	// Hier zum BMK noch die Ist-Position hinzufügen. Die Ist-Position wünschte sich nobilia. Das BMK bietet sich dafür an. Weitere Variablen in die Meldestruktur ist nicht möglich.
	IF IQ_stAchse.stMeldg.bEndlPosAngf
		OR bTestMeldAchs
	THEN
		IQ_stUniAnstgHMI.stAchsMeldHMI.sBMK :=
			CONCAT(I_sAktorBMK,
			CONCAT(' Istposition: ',TO_STRING(IQ_stAchse.fPosIstwert)));
	END_IF

	IQ_stUniAnstgHMI.stAchsMeldHMI.bMeldEndlPos				:= IQ_stAchse.stMeldg.bEndlPosAngf
																				OR bTestMeldAchs;			

	(**************************************************)
END_ACTION

END_FUNCTION_BLOCK

// POUs/UniBausteine/FB_UniAktrAnstg
(*
Beschreibung :	UniFB zur Hardwaresteuerung, Anzeige und Fehlermeldung in der Avalon HMI eines allgemeinen Aktors
					mit einem Überwachungseingang/Rückmeldung, ob auch eingeschaltet wurde.
					inkl. Handling - Handfunktinen
										- Meldefunktionen
										- Betriebsarten
										- Schutzbereiche
					Datentypen: ST_UniBaustein
									ST_UniAktrAnstg
					Ressourcen: GlobalVar_Allgemein
									GlobalVar_Farben
									AllgemeineParameter
TwinCat Vers.:	3.1.4024.25							
Erstellt		 :	Anlagentechnik Grp.11 (BECKHOFF AUTOMATION)
*)
FUNCTION_BLOCK FB_UniAktrAnstg
VAR_INPUT

	I_sStatName			:Tc2_System.T_MaxString;	// Aktueller Stationsname
	I_sAktorName		:Tc2_System.T_MaxString;	// Aktueller Aktorname von der Funktion des Aktors
	I_sAktorBMK1		:Tc2_System.T_MaxString;	// BMK - Rückmeldung

	I_bResHandFkt		:BOOL;	// Funktion-Reset für Grundstellungsablauf
	I_bZuwGrdstFkt		:BOOL;	// Funktion-Zuweisung Grundstellungsablauf
	I_bZuwAutomFkt		:BOOL;	// Funktion-Zuweisung Automatikablauf

	I_bAktrAbfrg		:BOOL;	// Abfrage z.B. Vakuum aufgebaut

	I_nSchutzBer		:INT;		// Schutzbereich => Betriebsart

	(*Optionale Funktionen*)													
	I_bResHdBetr		:BOOL;	// Ausschalten des Aktors beim Wechsel auf Handbetrieb
																						
	I_tLaufzVorg		:TIME:= T#5S;	(*Angepasste Meldelaufzeit*)	
	I_bVerrMeldg		:BOOL;	(*Meldungsausgabe Unterdrücken*)
																						
	I_bAnstgUng			:BOOL;	(*Ansteuerung Ungeschaltet*)	
	I_bAnstgInvt		:BOOL;	(*Ansteuerung Invertieren*)
	I_eAnstgDef			:E_AnstgArtUniAktr := eAktrAusEinschalt;	// Definition der Meldetexte und Anzeigetexte.
	
	I_sZuDef0			:Tc2_System.T_MaxString;	// eigene Definition für die linke Tasterbeschriftung
	I_sInDef0			:Tc2_System.T_MaxString;	// eigene Definition für die linke Tasterbeschriftung
	I_sZuDef1			:Tc2_System.T_MaxString;	// eigene Definition für die rechte Tasterbeschriftung
	I_sInDef1			:Tc2_System.T_MaxString;	// eigene Definition für die rechte Tasterbeschriftung

	I_stVarInfoBMK		:__SYSTEM.VAR_INFO;	// Optional: __VARINFO von einem Hardwareeingang. Kann I_sAktorBMK1 ersetzen. I_sAktorBMK1 ist aber dominant. Nicht im Aufruf verwenden => separate Zuweisung
END_VAR
VAR_IN_OUT

	IQ_stUniAnstgHMI	:ST_UniAktrAnstg;	// HMI-Strukturen

END_VAR
VAR_OUTPUT

	Q_bAktrAnstg		:BOOL;	// Ansteuerung z.B. Sauger Ein

END_VAR
VAR

	sTextHandFkt1		:ARRAY[0..1] OF STRING(20);				
	sTextHandFkt2		:ARRAY[0..1] OF STRING(20);					
	sTextHandFktX		:ARRAY[0..1] OF STRING(20);	// Zum Zwischenspeichern

	fbLfzMeldAusg		:FB_LaufzMeldgAktr;

	//Relevante Variablen zur Diagnose
	stUniAnstgFkt		:ST_UniBaustein;
END_VAR

	(*Uni.- Aktorenansteuerung*)
	
	(**************************************************)	
	(*Aufruf-Bereichskontrolle*)

	IF I_nSchutzBer <= 0 OR I_nSchutzBer > cAnzSchutzBer
		THEN
			IQ_stUniAnstgHMI.stMeldAusgHMI.sMeldText		:= 'I_nSchutzBer = 0 oder zu gross.';
			IQ_stUniAnstgHMI.stMeldAusgHMI.SourceName		:= I_sStatName;
			IQ_stUniAnstgHMI.stMeldAusgHMI.sAktorName		:= I_sAktorName;

			IF I_sAktorBMK1 <> ''
			THEN	// I_sAktorBMK1 ist beschrieben. Damit wird der String als BMK genommen
				IQ_stUniAnstgHMI.stMeldAusgHMI.sBMK	:= I_sAktorBMK1;
			ELSE	// Der Kommentar von VARINFO wird als BMK genommen
				IQ_stUniAnstgHMI.stMeldAusgHMI.sBMK	:= I_stVarInfoBMK.Comment;
			END_IF
			
			IQ_stUniAnstgHMI.stMeldAusgHMI.bMeldHinweis	:= TRUE;
			stUniAnstgFkt.nHandStat:= 256;	// Funktion sperren
			y_ZustAnzg();
			RETURN;
		ELSE
			IQ_stUniAnstgHMI.stMeldAusgHMI.bMeldHinweis	:= FALSE;
			IQ_stUniAnstgHMI.stMeldAusgHMI.sMeldText		:= '';
	END_IF

	(**************************************************)	
	(*Haendling Uni-Struktur*)

	a_Standard();

	(**************************************************)	
	(*Ausgänge zuweisen*)

	x_AusgZuw();
	
	(**************************************************)	
	(*Zustände anzeigen*)

	y_ZustAnzg();

	(**************************************************)	
	(*Meldungen ausgeben*)

	z_FehlMeld();
	
	(**************************************************)

ACTION a_Standard:
	(*Ansteuerungstyp "Standard" /z.B. Vakuumsauger...*)

	(*Verwendete Softkeytasten = 2 (s.Beispiel)*)

   (*       "Handfunktion"       /   "Softkeytaste 1"   /   "Softkeytaste 2"   *)
	(*                                                                          *) 
   (*------- Vakuumeinheit ------/_____ausschalten______/_____einschalten______*)
	
	(*Softkeyleiste.1		:Funktion ausschalten*)
	(*Softkeyleiste.2		:Funktion einschalten*)

	(*Hinweis:
	- Funktion wird durch "ResHdBetr" bei Betriebsartenwechsel zurückgenommen
	
	- Mit "LaufzVorg" kann die Meldelaufzeit angepasst werden (Default: 5sek)
	- Mit "VerrMeldg" wird die Meldeausgabe unterdrückt (eventl. Ablaufbedingt)
	
	- Bei "AnstgUng" bleiben die F-Ausgänge auch bei geöffn. Schutzbereich aktiv  
	- Bei "AnstgInvt" wird die Logik der Funktions-Ausgänge invertiert  
	*)

	(**************************************************)	

	stUniAnstgFkt.bHandAnw0:= IQ_stUniAnstgHMI.stHandFktHMI[1].bySwitch > 0;
	stUniAnstgFkt.bHandAnw1:= IQ_stUniAnstgHMI.stHandFktHMI[2].bySwitch > 0;
	
	IF arrBetrartAutomAktiv[I_nSchutzBer]
		OR I_bResHandFkt
		THEN
			stUniAnstgFkt.arrHandFkt[1]:= FALSE;
		ELSE
			IF arrBetrartAutomSpeichn[I_nSchutzBer]
				THEN
					IF NOT I_bResHdBetr THEN
						stUniAnstgFkt.arrHandFkt[1]:= stUniAnstgFkt.arrFktAusfg[1];
					END_IF
				ELSE
					IF NOT arrGrdstlgBetrAktiv[I_nSchutzBer]
						AND arrBetrartHandAktiv[I_nSchutzBer]
						THEN
							 IF stUniAnstgFkt.bHandAnw1 THEN
								 stUniAnstgFkt.arrHandFkt[1]:= TRUE;
							 END_IF
							 IF stUniAnstgFkt.bHandAnw0 THEN
								 stUniAnstgFkt.arrHandFkt[1]:= FALSE;
							 END_IF
					END_IF
			END_IF
	END_IF

	IF arrBetrartHandAktiv[I_nSchutzBer]
		THEN
			IF stUniAnstgFkt.arrHandFkt[1]
				THEN
					stUniAnstgFkt.nHandStat:= 2;	(*Handfunktion.2 aktiv*)
				ELSE
					stUniAnstgFkt.nHandStat:= 1;	(*Handfunktion.1 aktiv*)
			END_IF
		ELSE
			stUniAnstgFkt.nHandStat:= 256;		(*Funktion gesperrt*)
	END_IF

	(**************************************************)	

	IF arrBetrartHandAktiv[I_nSchutzBer]
		THEN
			stUniAnstgFkt.arrGrdstFkt[1]:= I_bZuwGrdstFkt;
		ELSE
			stUniAnstgFkt.arrGrdstFkt[1]:= FALSE;
   END_IF
	IF arrBetrartAutomAktiv[I_nSchutzBer] OR TRUE //ToDo
		THEN
			stUniAnstgFkt.arrAutomFkt[1]:= I_bZuwAutomFkt;
		ELSE
			stUniAnstgFkt.arrAutomFkt[1]:= FALSE;
   END_IF

	(**************************************************)	

	stUniAnstgFkt.arrFktAusfg[1]:= stUniAnstgFkt.arrGrdstFkt[1]
										  	 OR stUniAnstgFkt.arrHandFkt[1]
										    OR stUniAnstgFkt.arrAutomFkt[1];

	(**************************************************)
END_ACTION

ACTION x_AusgZuw:

	(**************************************************)	
	(*Ausgänge zuweisen*)

	Q_bAktrAnstg:= stUniAnstgFkt.arrFktAusfg[1]
					 	AND (arrAusgGruppeFrg[I_nSchutzBer]
				    	OR I_bAnstgUng)
					 	AND bVersEingAusgAnlagOk;

	(**************************************************)	
	(*Ausgänge invertieren*)

	IF I_bAnstgInvt THEN
		Q_bAktrAnstg:= NOT Q_bAktrAnstg;
	END_IF

	(**************************************************)
END_ACTION

ACTION y_ZustAnzg:
	
	(**************************************************)	
	(*Zustände anzeigen*)
	CASE I_eAnstgDef OF
eAktrDef0Def1,
eAktrDef1Def0:
						sTextHandFkt1[0]:= I_sZuDef0;
						sTextHandFkt1[1]:= I_sInDef0;
						sTextHandFkt2[0]:= I_sZuDef1;
						sTextHandFkt2[1]:= I_sInDef1;
	
eAktrAusEinschalt,
eAktrEinAusschalt:
						sTextHandFkt1[0]:= 'einschalten';
						sTextHandFkt1[1]:= 'eingeschaltet';
						sTextHandFkt2[0]:= 'ausschalten';
						sTextHandFkt2[1]:= 'ausgeschaltet';
eAktrAusEinfahr,
eAktrEinAusfahr:
						sTextHandFkt1[0]:= 'einfahren';
						sTextHandFkt1[1]:= 'eingefahren';
						sTextHandFkt2[0]:= 'ausfahren';
						sTextHandFkt2[1]:= 'ausgefahren';
eAktrHebenSenken,
eAktrSenkenHeben:
						sTextHandFkt1[0]:= 'senken';
						sTextHandFkt1[1]:= 'abgesenkt';
						sTextHandFkt2[0]:= 'heben';
						sTextHandFkt2[1]:= 'angehoben';
	END_CASE
	
	IF I_eAnstgDef >= 20 //Zuweisungen tauschen 
		THEN
			sTextHandFktX:= sTextHandFkt1; 
			sTextHandFkt1:= sTextHandFkt2;
			sTextHandFkt2:= sTextHandFktX;
	END_IF
	
	IF stUniAnstgFkt.nHandStat = 1	(*Handfunktion.1 aktiv*)
		THEN
			IQ_stUniAnstgHMI.stHandFktHMI[1].sColour:= cGruenAsString;
			IQ_stUniAnstgHMI.stHandFktHMI[1].sText:= sTextHandFkt1[1];
		ELSE
			IQ_stUniAnstgHMI.stHandFktHMI[1].sColour:= cDefaultAsString;
			IQ_stUniAnstgHMI.stHandFktHMI[1].sText:= sTextHandFkt1[0];
   END_IF
	IF stUniAnstgFkt.nHandStat = 2	(*Handfunktion.2 aktiv*)
		THEN		 
			IQ_stUniAnstgHMI.stHandFktHMI[2].sColour:= cGruenAsString;
			IQ_stUniAnstgHMI.stHandFktHMI[2].sText:= sTextHandFkt2[1];
		ELSE
			IQ_stUniAnstgHMI.stHandFktHMI[2].sColour:= cDefaultAsString;
			IQ_stUniAnstgHMI.stHandFktHMI[2].sText:= sTextHandFkt2[0];
   END_IF
	IF stUniAnstgFkt.nHandStat = 256	(*Funktion gesperrt*)
		THEN
			IQ_stUniAnstgHMI.stHandFktHMI[1].byStatus:=
			IQ_stUniAnstgHMI.stHandFktHMI[2].byStatus:= 1;
			IQ_stUniAnstgHMI.stHandFktHMI[1].sText:= sTextHandFkt1[0];
			IQ_stUniAnstgHMI.stHandFktHMI[2].sText:= sTextHandFkt2[0];
		ELSE
			IQ_stUniAnstgHMI.stHandFktHMI[1].byStatus:=
			IQ_stUniAnstgHMI.stHandFktHMI[2].byStatus:= 0;
   END_IF

	(**************************************************)
END_ACTION

ACTION z_FehlMeld:

	(**************************************************)	
	(*Meldungen ausgeben*)

	fbLfzMeldAusg.I_bLaufzAnstg1:=	(Q_bAktrAnstg
													AND NOT I_bAnstgInvt)
												OR (NOT Q_bAktrAnstg
													AND I_bAnstgInvt);
	fbLfzMeldAusg.I_bLaufzAbfrg1:=	I_bAktrAbfrg;

	fbLfzMeldAusg (I_bMeldgFreig	:= arrAusgGruppeFrg[I_nSchutzBer]
								   			AND bVersEingAusgAnlagOk
								   			AND NOT I_bVerrMeldg,
				  	   I_tLaufzDauer	:= I_tLaufzVorg);	(*Defaultwert = 5sek*)
		
	IQ_stUniAnstgHMI.stMeldAusgHMI.SourceID			:= 0;	// Nicht mehr verwendet
	IQ_stUniAnstgHMI.stMeldAusgHMI.SourceName			:= I_sStatName;
	IQ_stUniAnstgHMI.stMeldAusgHMI.sAktorName			:= I_sAktorName;
	
	IF I_sAktorBMK1 <> ''
	THEN	// I_sAktorBMK1 ist beschrieben. Damit wird der String als BMK genommen
		IQ_stUniAnstgHMI.stMeldAusgHMI.sBMK	:= I_sAktorBMK1;
	ELSE	// Der Kommentar von VARINFO wird als BMK genommen
		IQ_stUniAnstgHMI.stMeldAusgHMI.sBMK	:= I_stVarInfoBMK.Comment;
	END_IF

	IQ_stUniAnstgHMI.stMeldAusgHMI.bLfzMeldAusg		:= fbLfzMeldAusg.Q_bLaufzMeldg1
																		OR bTestMeldAktr; 
	IQ_stUniAnstgHMI.stMeldAusgHMI.bMeldHinweis		:= FALSE;	

		
	(**************************************************)
END_ACTION

END_FUNCTION_BLOCK

// POUs/UniBausteine/FB_UniAntrAnstg
(*
Beschreibung :	UniFB zur Handsteuerung, Anzeige und Fehlermeldungen in der Avalon-HMI eines Motors mit Schützsteuerung
					inkl. Handling - Handfunktinen
										- Meldefunktionen
										- Betriebsarten
										- Schutzbereiche
					Datentypen: ST_UniBaustein
									ST_UniAntrAnstg
					Ressourcen: GlobalVar_Allgemein
									GlobalVar_Farben
									AllgemeineParameter
TwinCat Vers.:	3.1.4024.25							
Erstellt		 :	Anlagentechnik Grp.11 (BECKHOFF AUTOMATION)
*)
FUNCTION_BLOCK FB_UniAntrAnstg
VAR_INPUT

	I_sSchaltSchr		:Tc2_System.T_MaxString;	// Aktueller Schaltschrank in dem die Schütze sitzen
	I_sAktorName		:Tc2_System.T_MaxString;	// Aktueller Aktorname von der Funktion des Motors
	I_sAktorBMK			:Tc2_System.T_MaxString;	// BMK vom Antrieb

	I_bResHandFkt		:BOOL;						// Funktion-Reset für Grundstellungsablauf. Alle Zuweisungen aus              
	I_arrZuwGrdstFkt	:ARRAY[0..1] OF BOOL;	// Funktion-Zuweisung Grundstellungsablauf: 0:RichtVrgZ 1:RichtVrgV
	I_arrZuwAutomFkt	:ARRAY[0..1] OF BOOL;	// Funktion-Zuweisung Automatikablauf: 0:RichtVrgZ 1:RichtVrgV

	I_bAbfrAbsgAntr	:BOOL;	// Abfrage z.B. Motorschutzschalter

	I_eAntriebTyp		:E_AntriebTyp;	// Antriebsfunktion

	I_sZuDef0			:Tc2_System.T_MaxString;	// eigene Definition für die linke Tasterbeschriftung
	I_sZuDef1			:Tc2_System.T_MaxString;	// eigene Definition für die rechte Tasterbeschriftung
	I_eAnstgDef			:E_AnstgArtUniAntr	:= eAntrAusEinschalt;			// Definition Ansteuerung

	I_nSchutzBer		:INT;		// Schutzbereich => Betriebsart

	// Optional /Antriebstyp Aggregat
	I_bResHdBetr		:BOOL;	// Auschalten des Motors beim Wechsel auf Handbetrieb
	// Optional /Antriebstyp Transport/Verstellung
	I_bVerrHdFktV		:BOOL;	// Sperren Handfunktion Richtung Vor	
	I_bVerrHdFktZ		:BOOL;	// Sperren Handfunktion Richtung Zurück
	// Optional /Antriebstyp Verstellung/Antriebstyp EilSchleich
	I_bEndlHdFktV		:BOOL;	// Endlage Sensor Richtung Vor		
	I_bEndlHdFktZ		:BOOL;	// Endlage Sensor Richtung Zurück

	I_stVarInfoBMK		:__SYSTEM.VAR_INFO;	// Optional: __VARINFO von einem Hardwareeingang. Kann I_sAktorBMK ersetzen. I_sAktorBMK ist aber dominant. Nicht im Aufruf verwenden => separate Zuweisung
END_VAR
VAR_IN_OUT
																								
	IQ_stUniAnstgHMI	:ST_UniAntrAnstg;	// HMI-Strukturen
																					
END_VAR
VAR_OUTPUT

	Q_bAnstNetzAntrV	:BOOL;	// Netzansteuerung Richtung Vor
	Q_bAnstNetzAntrZ	:BOOL;	// Netzansteuerung Richtung Zurück

END_VAR
VAR
																				
	rtrigHandFkt0		:R_TRIG;											
	rtrigHandFkt1		:R_TRIG;									

	//Relevante Variablen zur Diagnose
	stUniAnstgFkt		:ST_UniBaustein;
	
	sTextHandFkt1		:ARRAY[0..1] OF STRING(20);						
	sTextHandFkt2		:ARRAY[0..1] OF STRING(20);						
	sTextHandFktX		:ARRAY[0..1] OF STRING(20);	// Wird für den Vertausch der Texte benötigt.
END_VAR

	(*Uni.- Antriebsansteuerung*)
	
	(**************************************************)	
	(*Aufruf-Bereichskontrolle*)

	IF I_nSchutzBer <= 0 OR I_nSchutzBer > cAnzSchutzBer
		OR I_eAntriebTyp = E_AntriebTyp.eEilSchleich
		THEN
			IF I_nSchutzBer <= 0 OR I_nSchutzBer > cAnzSchutzBer
			THEN
				IQ_stUniAnstgHMI.stMeldAusgHMI.sMeldText		:= 'I_nSchutzBer = 0 oder zu gros.';
			ELSE
				IQ_stUniAnstgHMI.stMeldAusgHMI.sMeldText		:= 'I_eAntriebTyp = E_AntriebTyp.eEilSchleich gibt es hier nicht.';
			END_IF
			
			IQ_stUniAnstgHMI.stMeldAusgHMI.SourceName		:= I_sSchaltSchr;
			IQ_stUniAnstgHMI.stMeldAusgHMI.sAktorName		:= I_sAktorName;

			IF I_sAktorBMK <> ''
			THEN	// I_sAktorBMK ist beschrieben. Damit wird der String als BMK genommen
				IQ_stUniAnstgHMI.stMeldAusgHMI.sBMK	:= I_sAktorBMK;
			ELSE	// Der Kommentar von VARINFO wird als BMK genommen
				IQ_stUniAnstgHMI.stMeldAusgHMI.sBMK	:= I_stVarInfoBMK.Comment;
			END_IF
	
			IQ_stUniAnstgHMI.stMeldAusgHMI.bMeldHinweis	:= TRUE;

			stUniAnstgFkt.nHandStat:= 256;	// Funktion sperren
			y_ZustAnzg();
			RETURN;
		ELSE
			IQ_stUniAnstgHMI.stMeldAusgHMI.bMeldHinweis	:= FALSE;
			IQ_stUniAnstgHMI.stMeldAusgHMI.sMeldText		:= '';
	END_IF

	(**************************************************)	
	(*Haendling Uni-Struktur*)
	
	CASE I_eAntriebTyp OF
		 
1,5: (*Antriebstyp Aggregat*)
	
	a_Aggregat();

2:	(*Antriebstyp Transport*) 
	
	b_Transport();

3:	(*Antriebstyp Verstellg.*)

	c_Verstellg();
	
4:	(*Eilschleichachse gibts hier nicht*)

	RETURN;

   END_CASE

	(**************************************************)	
	(*Ausgänge zuweisen*)

	x_AusgZuw();
	
	(**************************************************)	
	(*Zustände anzeigen*)

	y_ZustAnzg();

	(**************************************************)	
	(*Meldungen ausgeben*)

	z_FehlMeld();
	
	(**************************************************)

ACTION a_Aggregat:
	(*Antriebstyp "Aggregat" /z.B. Bohraggregate...*)

	(*Verwendete Softkeytasten = 5 (s.Beispiel)*)

   (*       "Handfunktion"       /   "Softkeytaste 1"   /   "Softkeytaste 2"   /   "Softkeytaste 3"   /   "Softkeytaste 4"   /   "Softkeytaste 5"   *)
	(*                                                                          															  								 *) 
   (*------- Bohraggregat -------/_____ausschalten______/_____einschalten______/_________Frei_________/_________Frei_________/_________Frei_________*)

	(*Softkeyleiste.1		:Funktion ausschalten*)
	(*Softkeyleiste.2		:Funktion einschalten*)
	(*Softkeyleiste.3		:Platzhalter			*)
	(*Softkeyleiste.4		:Platzhalter			*)
	(*Softkeyleiste.5		:Platzhalter			*)

	(*Hinweis:
	- Funktion wird durch "ResHdBetr" bei Betriebsartenwechsel zurückgenommen
	*)

	(**************************************************)	

	stUniAnstgFkt.bHandAnw0:= IQ_stUniAnstgHMI.stHandFktHMI[1].bySwitch > 0;
	stUniAnstgFkt.bHandAnw1:= IQ_stUniAnstgHMI.stHandFktHMI[2].bySwitch > 0;
	
	IF arrBetrartAutomAktiv[I_nSchutzBer]
		OR I_bResHandFkt
		THEN
			stUniAnstgFkt.arrHandFkt[1]:= FALSE;
		ELSE
			IF arrBetrartAutomSpeichn[I_nSchutzBer]
				THEN
					IF NOT I_bResHdBetr THEN
						stUniAnstgFkt.arrHandFkt[1]:= stUniAnstgFkt.arrFktAusfg[1];
					END_IF
				ELSE
					IF NOT arrGrdstlgBetrAktiv[I_nSchutzBer]
						AND arrBetrartHandAktiv[I_nSchutzBer]
						THEN
							 IF stUniAnstgFkt.bHandAnw1 THEN
								 stUniAnstgFkt.arrHandFkt[1]:= TRUE;
							 END_IF
							 IF stUniAnstgFkt.bHandAnw0 THEN
								 stUniAnstgFkt.arrHandFkt[1]:= FALSE;
							 END_IF
					END_IF
			END_IF
	END_IF

	IF arrBetrartHandAktiv[I_nSchutzBer]
		THEN
			IF stUniAnstgFkt.arrHandFkt[1]
				THEN
					stUniAnstgFkt.nHandStat:= 2;	(*Handfunktion.2 aktiv*)
				ELSE
					stUniAnstgFkt.nHandStat:= 1;	(*Handfunktion.1 aktiv*)
			END_IF
		ELSE
			stUniAnstgFkt.nHandStat:= 256;		(*Funktion gesperrt*)
	END_IF

	(**************************************************)	

	IF arrBetrartHandAktiv[I_nSchutzBer]
		THEN
			stUniAnstgFkt.arrGrdstFkt[1]:= I_arrZuwGrdstFkt[1];
		ELSE
			stUniAnstgFkt.arrGrdstFkt[1]:= FALSE;
   END_IF
	IF arrBetrartAutomAktiv[I_nSchutzBer] OR TRUE //ToDo
		THEN
			stUniAnstgFkt.arrAutomFkt[1]:= I_arrZuwAutomFkt[1];
		ELSE
			stUniAnstgFkt.arrAutomFkt[1]:= FALSE;
   END_IF

	(**************************************************)	

	stUniAnstgFkt.arrFktAusfg[1]:= stUniAnstgFkt.arrGrdstFkt[1]
											 OR stUniAnstgFkt.arrHandFkt[1]
											 OR stUniAnstgFkt.arrAutomFkt[1];

	(**************************************************)
END_ACTION

ACTION b_Transport:
	(*Antriebstyp "Transport" /z.B. Förderantriebe...*)

	(*Verwendete Softkeytasten = 5 (s.Beispiel)*)

   (*       "Handfunktion"       /   "Softkeytaste 1"   /   "Softkeytaste 2"   /   "Softkeytaste 3"   /   "Softkeytaste 4"   /   "Softkeytaste 5"   *)
	(*                                                                          															  								 *) 
	(*----- Transportantrieb -----/_einschalten (zurück)_/___einschalten (vor)__/_________Frei_________/_________Frei_________/_________Frei_________*)

	(*Softkeyleiste.1		:Funktion ein.-ausschalten Reversierend*)
	(*Softkeyleiste.2		:Funktion ein.-ausschalten             *)
	(*Softkeyleiste.3		:Platzhalter				 					*)
	(*Softkeyleiste.4		:Platzhalter				 					*)
	(*Softkeyleiste.5		:Platzhalter				 					*)

	(*Hinweis:
	- Funktion wird durch "VerrHdFkt" gesperrt (z.B. kein Reversierbetrieb...)
	*)

	(**************************************************)	

	stUniAnstgFkt.bHandAnw0:= IQ_stUniAnstgHMI.stHandFktHMI[1].bySwitch > 0;
	stUniAnstgFkt.bHandAnw1:= IQ_stUniAnstgHMI.stHandFktHMI[2].bySwitch > 0;
	
	IF arrBetrartAutomAktiv[I_nSchutzBer]
		OR I_bResHandFkt
		THEN
			stUniAnstgFkt.arrHandFkt[0]:=
			stUniAnstgFkt.arrHandFkt[1]:= FALSE;
		ELSE
			IF NOT arrBetrartAutomSpeichn[I_nSchutzBer]
				THEN
					IF NOT arrGrdstlgBetrAktiv[I_nSchutzBer]
						THEN
							 rtrigHandFkt1 (CLK:= stUniAnstgFkt.bHandAnw1);
							 IF rtrigHandFkt1.Q THEN
								 stUniAnstgFkt.arrHandFkt[1]:= NOT stUniAnstgFkt.arrHandFkt[1];
							 END_IF
							 IF NOT arrBetrartHandAktiv[I_nSchutzBer]
								 OR stUniAnstgFkt.arrHandFkt[0]
								 OR I_bVerrHdFktV THEN
								 stUniAnstgFkt.arrHandFkt[1]:= FALSE;
							 END_IF
	 
							 rtrigHandFkt0 (CLK:= stUniAnstgFkt.bHandAnw0);
							 IF rtrigHandFkt0.Q THEN
								 stUniAnstgFkt.arrHandFkt[0]:= NOT stUniAnstgFkt.arrHandFkt[0];
							 END_IF
							 IF NOT arrBetrartHandAktiv[I_nSchutzBer]
								 OR stUniAnstgFkt.arrHandFkt[1]
								 OR I_bVerrHdFktZ THEN
								 stUniAnstgFkt.arrHandFkt[0]:= FALSE;
							 END_IF
					END_IF
			END_IF
	END_IF

	IF arrBetrartHandAktiv[I_nSchutzBer]
		THEN
			stUniAnstgFkt.nHandStat:= 0;			(*Funktion freigegeben*)
			IF stUniAnstgFkt.arrHandFkt[1]
				THEN
					stUniAnstgFkt.nHandStat:= 2;	(*Handfunktion.2 aktiv*)
			END_IF
			IF stUniAnstgFkt.arrHandFkt[0]
				THEN
					stUniAnstgFkt.nHandStat:= 1;	(*Handfunktion.1 aktiv*)
			END_IF
		ELSE
			stUniAnstgFkt.nHandStat:= 256;		(*Funktion gesperrt*)
	END_IF

	(**************************************************)	

	IF arrBetrartHandAktiv[I_nSchutzBer]
		THEN
			stUniAnstgFkt.arrGrdstFkt[0]:= I_arrZuwGrdstFkt[0];
			stUniAnstgFkt.arrGrdstFkt[1]:= I_arrZuwGrdstFkt[1];
		ELSE
			stUniAnstgFkt.arrGrdstFkt[0]:= 
			stUniAnstgFkt.arrGrdstFkt[1]:= FALSE;
   END_IF
	IF arrBetrartAutomAktiv[I_nSchutzBer] OR TRUE //ToDo
		THEN
			stUniAnstgFkt.arrAutomFkt[0]:= I_arrZuwAutomFkt[0];
			stUniAnstgFkt.arrAutomFkt[1]:= I_arrZuwAutomFkt[1];
		ELSE
			stUniAnstgFkt.arrAutomFkt[0]:= 
			stUniAnstgFkt.arrAutomFkt[1]:= FALSE;
   END_IF

	(**************************************************)	

	stUniAnstgFkt.arrFktAusfg[0]:= stUniAnstgFkt.arrGrdstFkt[0]
											 OR stUniAnstgFkt.arrHandFkt[0]
											 OR stUniAnstgFkt.arrAutomFkt[0];

	stUniAnstgFkt.arrFktAusfg[1]:= stUniAnstgFkt.arrGrdstFkt[1]
											 OR stUniAnstgFkt.arrHandFkt[1]
											 OR stUniAnstgFkt.arrAutomFkt[1];

	(**************************************************)
END_ACTION

ACTION c_Verstellg:
	(*Antriebstyp "Verstellg." /z.B. Zustellantriebe mit Wendeschütz...*)

	(*Verwendete Softkeytasten = 5 (s.Beispiel)*)

   (*       "Handfunktion"       /   "Softkeytaste 1"   /   "Softkeytaste 2"   /   "Softkeytaste 3"   /   "Softkeytaste 4"   /   "Softkeytaste 5"   *)
	(*                                                                          															  								 *) 
	(*----- Verstellantrieb ------/_____zurückfahren_____/_______vorfahren______/_________Frei_________/_________Frei_________/_________Frei_________*)

	(*Softkeyleiste.1		:Funktion ein.-ausschalten Reversierend*)
	(*Softkeyleiste.2		:Funktion ein.-ausschalten             *)
	(*Softkeyleiste.3		:Platzhalter				 					*)
	(*Softkeyleiste.4		:Platzhalter				 					*)
	(*Softkeyleiste.5		:Platzhalter				 					*)

	(*Hinweis:
	- Funktion wird durch "VerrHdFkt" gesperrt (z.B. bei Überstandserkennung...)
	- Funktion wird durch "EndlHdFkt/VerzHdFkt" zurückgenommen bzw. umgeschaltet
	*)
	
	(**************************************************)	

	stUniAnstgFkt.bHandAnw0:= IQ_stUniAnstgHMI.stHandFktHMI[1].bySwitch > 0;
	stUniAnstgFkt.bHandAnw1:= IQ_stUniAnstgHMI.stHandFktHMI[2].bySwitch > 0;
	
	IF arrBetrartAutomAktiv[I_nSchutzBer]
		OR I_bResHandFkt
		THEN
			stUniAnstgFkt.arrHandFkt[0]:=
			stUniAnstgFkt.arrHandFkt[1]:= FALSE;
		ELSE
			IF NOT arrBetrartAutomSpeichn[I_nSchutzBer]
				THEN
					IF NOT arrGrdstlgBetrAktiv[I_nSchutzBer]
						THEN
							 rtrigHandFkt1 (CLK:= stUniAnstgFkt.bHandAnw1);
							 IF rtrigHandFkt1.Q THEN
								 stUniAnstgFkt.arrHandFkt[1]:= NOT stUniAnstgFkt.arrHandFkt[1];
							 END_IF
							 IF NOT arrBetrartHandAktiv[I_nSchutzBer]
								 OR stUniAnstgFkt.arrHandFkt[0]
								 OR I_bVerrHdFktV OR NOT I_bEndlHdFktV THEN
								 stUniAnstgFkt.arrHandFkt[1]:= FALSE;
							 END_IF
	 
							 rtrigHandFkt0 (CLK:= stUniAnstgFkt.bHandAnw0);
							 IF rtrigHandFkt0.Q THEN
								 stUniAnstgFkt.arrHandFkt[0]:= NOT stUniAnstgFkt.arrHandFkt[0];
							 END_IF
							 IF NOT arrBetrartHandAktiv[I_nSchutzBer]
								 OR stUniAnstgFkt.arrHandFkt[1]
								 OR I_bVerrHdFktZ OR NOT I_bEndlHdFktZ THEN
								 stUniAnstgFkt.arrHandFkt[0]:= FALSE;
							 END_IF
					END_IF
			END_IF
	END_IF

	IF arrBetrartHandAktiv[I_nSchutzBer]
		THEN
			stUniAnstgFkt.nHandStat:= 0;			(*Funktion freigegeben*)
			IF stUniAnstgFkt.arrHandFkt[1]
				THEN
					stUniAnstgFkt.nHandStat:= 2;	(*Handfunktion.2 aktiv*)
			END_IF
			IF stUniAnstgFkt.arrHandFkt[0]
				THEN
					stUniAnstgFkt.nHandStat:= 1;	(*Handfunktion.1 aktiv*)
			END_IF
		ELSE
			stUniAnstgFkt.nHandStat:= 256;		(*Funktion gesperrt*)
	END_IF

	(**************************************************)	

	IF arrBetrartHandAktiv[I_nSchutzBer]
		THEN
			stUniAnstgFkt.arrGrdstFkt[0]:= I_arrZuwGrdstFkt[0];
			stUniAnstgFkt.arrGrdstFkt[1]:= I_arrZuwGrdstFkt[1];
		ELSE
			stUniAnstgFkt.arrGrdstFkt[0]:= 
			stUniAnstgFkt.arrGrdstFkt[1]:= FALSE;
   END_IF
	IF arrBetrartAutomAktiv[I_nSchutzBer] OR TRUE //ToDo
		THEN
			stUniAnstgFkt.arrAutomFkt[0]:= I_arrZuwAutomFkt[0];
			stUniAnstgFkt.arrAutomFkt[1]:= I_arrZuwAutomFkt[1];
		ELSE
			stUniAnstgFkt.arrAutomFkt[0]:= 
			stUniAnstgFkt.arrAutomFkt[1]:= FALSE;
   END_IF

	(**************************************************)	

	stUniAnstgFkt.arrFktAusfg[0]:= stUniAnstgFkt.arrGrdstFkt[0]
											 OR stUniAnstgFkt.arrHandFkt[0]
											 OR stUniAnstgFkt.arrAutomFkt[0];

	stUniAnstgFkt.arrFktAusfg[1]:= stUniAnstgFkt.arrGrdstFkt[1]
											 OR stUniAnstgFkt.arrHandFkt[1]
											 OR stUniAnstgFkt.arrAutomFkt[1];

	(**************************************************)
END_ACTION

ACTION x_AusgZuw:

	(**************************************************)	
	(*Ausgänge zuweisen*)

	Q_bAnstNetzAntrV:= stUniAnstgFkt.arrFktAusfg[1]
						 	 AND NOT Q_bAnstNetzAntrZ
						 	 AND arrAntrGruppeFrg[I_nSchutzBer]
						 	 AND I_bAbfrAbsgAntr
						 	 AND bVersEingAusgSchaltsOk;

	Q_bAnstNetzAntrZ:= stUniAnstgFkt.arrFktAusfg[0]
						 	 AND NOT Q_bAnstNetzAntrV
						 	 AND arrAntrGruppeFrg[I_nSchutzBer]
						 	 AND I_bAbfrAbsgAntr
						 	 AND bVersEingAusgSchaltsOk;

	(**************************************************)
END_ACTION

ACTION y_ZustAnzg:



// die Zahlen 0-8 sind wegen der Abwärtskompatibiliät noch drin.
CASE I_eAnstgDef OF
	
eAntrDef0Def1,eAntrDef1Def0:
	sTextHandFkt1[0]:= I_sZuDef0;
	sTextHandFkt2[0]:= I_sZuDef1;
eAntrEinAusschalt,eAntrAusEinschalt:
	sTextHandFkt1[0]:= 'ausschalten';
	sTextHandFkt2[0]:= 'einschalten';
eAntrEinAusfahr,eAntrAusEinfahr:
	sTextHandFkt1[0]:= 'ausfahren';
	sTextHandFkt2[0]:= 'einfahren';
eAntrHebenSenken,eAntrSenkenHeben:
	sTextHandFkt1[0]:= 'senken';
	sTextHandFkt2[0]:= 'heben';
eAntrVorZurueck,eAntrZurueckVor:
	sTextHandFkt1[0]:= 'zurückfahren';
	sTextHandFkt2[0]:= 'vorfahren';
END_CASE
	
IF I_eAnstgDef >= 50 //Zuweisungen tauschen 
	THEN
		sTextHandFktX:= sTextHandFkt1; 
		sTextHandFkt1:= sTextHandFkt2;
		sTextHandFkt2:= sTextHandFktX;
END_IF
	
	
	(**************************************************)	
	(*Zustände anzeigen*)

	CASE I_eAntriebTyp OF

1:	(*Antriebstyp Aggregat*)
	
	IF stUniAnstgFkt.nHandStat = 1	(*Handfunktion.1 aktiv*)
		THEN
			IQ_stUniAnstgHMI.stHandFktHMI[1].sColour:= cGruenAsString; //eventl.: cRot;
			IQ_stUniAnstgHMI.stHandFktHMI[2].sColour:= cDefaultAsString;
			IQ_stUniAnstgHMI.stHandFktHMI[1].sText:= sTextHandFkt1[0];
			IQ_stUniAnstgHMI.stHandFktHMI[2].sText:= sTextHandFkt2[0];
   END_IF
	IF stUniAnstgFkt.nHandStat = 2	(*Handfunktion.2 aktiv*)
		THEN		 
			IQ_stUniAnstgHMI.stHandFktHMI[1].sColour:= cDefaultAsString;
			IQ_stUniAnstgHMI.stHandFktHMI[2].sColour:= cGruenAsString;
			IQ_stUniAnstgHMI.stHandFktHMI[1].sText:= sTextHandFkt1[0];
			IQ_stUniAnstgHMI.stHandFktHMI[2].sText:= sTextHandFkt2[0];
   END_IF
	IQ_stUniAnstgHMI.stHandFktHMI[3].sColour:= cDefaultAsString;
	IQ_stUniAnstgHMI.stHandFktHMI[3].sText:= ' ';
	IQ_stUniAnstgHMI.stHandFktHMI[4].sColour:= cDefaultAsString;
	IQ_stUniAnstgHMI.stHandFktHMI[4].sText:= ' ';
	IQ_stUniAnstgHMI.stHandFktHMI[5].sColour:= cDefaultAsString;
	IQ_stUniAnstgHMI.stHandFktHMI[5].sText:= ' ';
	IF stUniAnstgFkt.nHandStat = 256	(*Funktion gesperrt*)
		THEN
			IQ_stUniAnstgHMI.stHandFktHMI[1].sText:= 'ausgeschaltet';
			IQ_stUniAnstgHMI.stHandFktHMI[2].sText:= sTextHandFkt2[0];
			IQ_stUniAnstgHMI.stHandFktHMI[1].sColour:=
			IQ_stUniAnstgHMI.stHandFktHMI[2].sColour:=cDefaultAsString;
			IQ_stUniAnstgHMI.stHandFktHMI[1].byStatus:=
			IQ_stUniAnstgHMI.stHandFktHMI[2].byStatus:=
			IQ_stUniAnstgHMI.stHandFktHMI[3].byStatus:=
			IQ_stUniAnstgHMI.stHandFktHMI[4].byStatus:=
			IQ_stUniAnstgHMI.stHandFktHMI[5].byStatus:= 1;
		ELSE
			IQ_stUniAnstgHMI.stHandFktHMI[1].byStatus:=
			IQ_stUniAnstgHMI.stHandFktHMI[2].byStatus:=
			IQ_stUniAnstgHMI.stHandFktHMI[3].byStatus:=
			IQ_stUniAnstgHMI.stHandFktHMI[4].byStatus:=
			IQ_stUniAnstgHMI.stHandFktHMI[5].byStatus:= 0;
   END_IF

2:	(*Antriebstyp Transport*) 
	
	IF stUniAnstgFkt.nHandStat = 1	(*Handfunktion.1 aktiv*)
		THEN
			IQ_stUniAnstgHMI.stHandFktHMI[1].sColour:= cGruenAsString;
			IQ_stUniAnstgHMI.stHandFktHMI[1].sText:= sTextHandFkt1[0];
		ELSE
			IQ_stUniAnstgHMI.stHandFktHMI[1].sColour:= cDefaultAsString;
			IQ_stUniAnstgHMI.stHandFktHMI[1].sText:= sTextHandFkt1[0];
			IF stUniAnstgFkt.nHandStat = 2 THEN
				IQ_stUniAnstgHMI.stHandFktHMI[1].sText:= ' ';
			END_IF
   END_IF
	IF stUniAnstgFkt.nHandStat = 2	(*Handfunktion.2 aktiv*)
		THEN		 
			IQ_stUniAnstgHMI.stHandFktHMI[2].sColour:= cGruenAsString;
			IQ_stUniAnstgHMI.stHandFktHMI[2].sText:= sTextHandFkt2[0];
		ELSE
			IQ_stUniAnstgHMI.stHandFktHMI[2].sColour:= cDefaultAsString;
			IQ_stUniAnstgHMI.stHandFktHMI[2].sText:= sTextHandFkt2[0];
			IF stUniAnstgFkt.nHandStat = 1 THEN
				IQ_stUniAnstgHMI.stHandFktHMI[2].sText:= ' ';
			END_IF
   END_IF
	IQ_stUniAnstgHMI.stHandFktHMI[3].sColour:= cDefaultAsString;
	IQ_stUniAnstgHMI.stHandFktHMI[3].sText:= ' ';
	IQ_stUniAnstgHMI.stHandFktHMI[4].sColour:= cDefaultAsString;
	IQ_stUniAnstgHMI.stHandFktHMI[4].sText:= ' ';
	IQ_stUniAnstgHMI.stHandFktHMI[5].sColour:= cDefaultAsString;
	IQ_stUniAnstgHMI.stHandFktHMI[5].sText:= ' ';
	IF stUniAnstgFkt.nHandStat = 256	(*Funktion gesperrt*)
		THEN
			IQ_stUniAnstgHMI.stHandFktHMI[1].sText:= sTextHandFkt1[0];
			IQ_stUniAnstgHMI.stHandFktHMI[2].sText:= sTextHandFkt2[0];
			IQ_stUniAnstgHMI.stHandFktHMI[1].sColour:=
			IQ_stUniAnstgHMI.stHandFktHMI[2].sColour:= cDefaultAsString;
			IQ_stUniAnstgHMI.stHandFktHMI[1].byStatus:=
			IQ_stUniAnstgHMI.stHandFktHMI[2].byStatus:=
			IQ_stUniAnstgHMI.stHandFktHMI[3].byStatus:=
			IQ_stUniAnstgHMI.stHandFktHMI[4].byStatus:=
			IQ_stUniAnstgHMI.stHandFktHMI[5].byStatus:= 1;
		ELSE
			IQ_stUniAnstgHMI.stHandFktHMI[1].byStatus:=
			IQ_stUniAnstgHMI.stHandFktHMI[2].byStatus:=
			IQ_stUniAnstgHMI.stHandFktHMI[3].byStatus:=
			IQ_stUniAnstgHMI.stHandFktHMI[4].byStatus:=
			IQ_stUniAnstgHMI.stHandFktHMI[5].byStatus:= 0;
   END_IF

3:	(*Antriebstyp Verstellg.*)
	
	IF stUniAnstgFkt.nHandStat = 1	(*Handfunktion.1 aktiv*)
		THEN
			IQ_stUniAnstgHMI.stHandFktHMI[1].sColour:= cGruenAsString;
			IQ_stUniAnstgHMI.stHandFktHMI[1].sText:= sTextHandFkt1[0];
		ELSE
			IQ_stUniAnstgHMI.stHandFktHMI[1].sColour:= cDefaultAsString;
			IQ_stUniAnstgHMI.stHandFktHMI[1].sText:= sTextHandFkt1[0];
   END_IF
	IF stUniAnstgFkt.nHandStat = 2	(*Handfunktion.2 aktiv*)
		THEN		 
			IQ_stUniAnstgHMI.stHandFktHMI[2].sColour:= cGruenAsString;
			IQ_stUniAnstgHMI.stHandFktHMI[2].sText:= sTextHandFkt2[0];
		ELSE
			IQ_stUniAnstgHMI.stHandFktHMI[2].sColour:= cDefaultAsString;
			IQ_stUniAnstgHMI.stHandFktHMI[2].sText:= sTextHandFkt2[0];
   END_IF
	IQ_stUniAnstgHMI.stHandFktHMI[3].sColour:= cDefaultAsString;
	IQ_stUniAnstgHMI.stHandFktHMI[3].sText:= ' ';
	IQ_stUniAnstgHMI.stHandFktHMI[4].sColour:= cDefaultAsString;
	IQ_stUniAnstgHMI.stHandFktHMI[4].sText:= ' ';
	IQ_stUniAnstgHMI.stHandFktHMI[5].sColour:= cDefaultAsString;
	IQ_stUniAnstgHMI.stHandFktHMI[5].sText:= ' ';
	IF stUniAnstgFkt.nHandStat = 256	(*Funktion gesperrt*)
		THEN
			IQ_stUniAnstgHMI.stHandFktHMI[1].sText:= sTextHandFkt1[0];
			IQ_stUniAnstgHMI.stHandFktHMI[2].sText:= sTextHandFkt2[0];
			IQ_stUniAnstgHMI.stHandFktHMI[1].sColour:=
			IQ_stUniAnstgHMI.stHandFktHMI[2].sColour:= cDefaultAsString;
			IQ_stUniAnstgHMI.stHandFktHMI[1].byStatus:=
			IQ_stUniAnstgHMI.stHandFktHMI[2].byStatus:=
			IQ_stUniAnstgHMI.stHandFktHMI[3].byStatus:=
			IQ_stUniAnstgHMI.stHandFktHMI[4].byStatus:=
			IQ_stUniAnstgHMI.stHandFktHMI[5].byStatus:= 1;
		ELSE
			IQ_stUniAnstgHMI.stHandFktHMI[1].byStatus:=
			IQ_stUniAnstgHMI.stHandFktHMI[2].byStatus:=
			IQ_stUniAnstgHMI.stHandFktHMI[3].byStatus:=
			IQ_stUniAnstgHMI.stHandFktHMI[4].byStatus:=
			IQ_stUniAnstgHMI.stHandFktHMI[5].byStatus:= 0;
   END_IF

   END_CASE

	(**************************************************)
END_ACTION

ACTION z_FehlMeld:

	(**************************************************)	
	(*Meldungen ausgeben*)

	IQ_stUniAnstgHMI.stMeldAusgHMI.SourceID		:= 0;	// Nicht mehr verwendet
	IQ_stUniAnstgHMI.stMeldAusgHMI.SourceName		:= I_sSchaltSchr;
	IQ_stUniAnstgHMI.stMeldAusgHMI.sAktorName		:= I_sAktorName;

	IF I_sAktorBMK <> ''
	THEN	// I_sAktorBMK ist beschrieben. Damit wird der String als BMK genommen
		IQ_stUniAnstgHMI.stMeldAusgHMI.sBMK	:= I_sAktorBMK;
	ELSE	// Der Kommentar von VARINFO wird als BMK genommen
		IQ_stUniAnstgHMI.stMeldAusgHMI.sBMK	:= I_stVarInfoBMK.Comment;
	END_IF

	IQ_stUniAnstgHMI.stMeldAusgHMI.bMeldNichtBtb	:= (arrAntrGruppeFrg[I_nSchutzBer]
																		AND NOT I_bAbfrAbsgAntr
																		AND bVersEingAusgSchaltsOk)
																	OR bTestMeldAntr;

	(**************************************************)
END_ACTION

END_FUNCTION_BLOCK

// POUs/UniBausteine/FB_UniAntrAnstgSEW
(*
Beschreibung :	SEW-FU-Steuerung  über Prozessabbild mit der FSE24B-Schnittstelle.
					inkl. Handling - Handfunktinen
										- Meldefunktionen
										- Betriebsarten
										- Schutzbereiche
					Datentypen: ST_UniBaustein
									ST_UniAntrAnstg
					Ressourcen: GlobalVar_Allgemein
									GlobalVar_Farben
									AllgemeineParameter
									ST_NcAchsen
									Tc2_MC2.AXIS_REF
TwinCat Vers.:	3.1.4024.25							
Erstellt		 :	Anlagentechnik Grp.11 (BECKHOFF AUTOMATION)
*)
FUNCTION_BLOCK FB_UniAntrAnstgSEW
VAR_INPUT

	I_sSchaltSchr		:Tc2_System.T_MaxString;	(*Aktueller Schaltschrank*)
	I_sStatName			:Tc2_System.T_MaxString;	(*Aktueller Stationsname*)
	I_sAktorName		:Tc2_System.T_MaxString;	(*Aktueller Aktorname*)
	I_sAktorBMK			:Tc2_System.T_MaxString;	(*BMK - Betriebsbereit*)

	I_bResHandFkt		:BOOL;						(*Fkt.-Reset für Grdstlg.-ablauf*)
	I_arrZuwGrdstFkt	:ARRAY[0..2] OF BOOL;	(*Fkt.-Zuweisung Grdstlg.-ablauf*)
	I_arrZuwAutomFkt	:ARRAY[0..2] OF BOOL;	(*Fkt.-Zuweisung Automatikablauf*)
															(*0:RichtVrgZ 1:RichtVrgV 2:SollwVrg*)

	I_stSEWInput		:ST_SEWInput;	// SEW-Eingänge
																					
	I_bUmrReset			:BOOL;	// Umrichter-Reset
																					
	I_eAntriebTyp		:E_AntriebTyp;	// Antriebsfunktion

	I_RefAchse			:REFERENCE TO ST_NcAchsen;	// Verweis zur arrNcAchsen-Strucktur. Bei einer Eil-Schleichachse einfach zuweisen.
	I_RefAxis			:REFERENCE TO Tc2_MC2.AXIS_REF;	// Verweis zur arrAxisRef-Strucktur. Bei einer Eil-Schleichachse einfach zuweisen.

	I_nAntrEinsGrp		:INT;		// Aktuelle Netzeinschaltgruppe
	I_nSchutzBer		:INT;		// Schutzbereich => Betriebsart

	I_fSollwMinUmr		:LREAL;	(*Drehzahl.-Geschwindigkeitsuntergrenze*)
	I_fSollwMaxUmr		:LREAL;	(*Drehzahl.-Geschwindigkeitsobergrenze. Kann aber auch über Maschinenparameter vorgegeben werden. Der Eingang ist aber Dominant.*)
	I_fSollwVrgUmr		:LREAL;	(*Drehzahl.-Geschwindigkeitsvorgabe*)
									  	(*Einheit: Prozentual (SollwMax = Nmax)*)
	I_fRampVrgBUmr		:LREAL;	(*Vorgabe Beschleunigungsrampe*)
	I_fRampVrgVUmr		:LREAL;	(*Vorgabe Verzögerungsrampe*)
									  	(*Einheit: mSek*)

	// Optional /Antriebstyp Aggregat
	I_bResHdBetr		:BOOL;	// Auschalten des Motors beim Wechsel auf Handbetrieb
	// Optional /Antriebstyp Transport/Verstellung
	I_bVerrHdFktV		:BOOL;	// Sperren Handfunktion Richtung Vor	
	I_bVerrHdFktZ		:BOOL;	// Sperren Handfunktion Richtung Zurück
	// Optional /Antriebstyp Verstellung/Antriebstyp EilSchleich
	I_bEndlHdFktV		:BOOL;	// Endlage Sensor Richtung Vor		
	I_bEndlHdFktZ		:BOOL;	// Endlage Sensor Richtung Zurück	
	I_bVerzHdFktV		:BOOL;	// Verzögerung Sensor Richtung Vor	
	I_bVerzHdFktZ		:BOOL;	// Verzögerung Sensor Richtung Zurück

	I_bExtReglFrg		:BOOL:= TRUE; // Externes Freigabesignal

	I_bAnwEinlZykl		:BOOL;	// Anwahl Erstinbetriebn.-Einlaufzyklus

	I_bStandbyBetr		:BOOL;	// Antrieb im Standby-Betrieb. Kann statt I_arrZuwAutomFkt[1] zur Hochlaufphase genutzt werden.
	
	I_tLaufzeitMeld	:TIME := T#10S; // Zeit bis zur Laufzeitmeldung

{attribute 'hide'}
	I_arrBetrZyklPhase	:ARRAY[1..4] OF TIME	:= [T#1M,T#1M,T#1M,T#1M];	// Zeiten für das Warmlauf im Betrieb 1-3 ist Warmlaufen 4 ist Warmhalten
{attribute 'hide'}
	I_arrBetrZyklDrehz	:ARRAY[1..4] OF LREAL	:= [50,75,100,20];	// Drehzahlen in % für das Warmlauf im Betrieb 1-3 ist Warmlaufen 4 ist Warmhalten
{attribute 'hide'}	
	I_tPause				:TIME := T#15M;
	
	I_stVarInfoBMK		:__SYSTEM.VAR_INFO;	// Optional: __VARINFO von dem Hardwareeingang I_stSEWInput oder I_stSEWOutput. Kann I_sAktorBMK ersetzen. I_sAktorBMK ist aber dominant. Nicht im Aufruf verwenden => separate Zuweisung
END_VAR
VAR_IN_OUT

	IQ_stUniAnstgHMI	:ST_UniAntrAnstg;	(*HMI-Strukturen*)

END_VAR
VAR_OUTPUT
																						
	Q_bAbfrStatUmr		:BOOL;	(*Statusabfrage Umrichter*)			
	Q_nAbfrUmrDrehz	:INT;		(*Umrichterabfrage Istdrehzahl*)		
	Q_nAbfrUmrStrom	:INT;		(*Umrichterabfrage Iststrom/%*)	
	Q_bUmrDrehzNnull	:BOOL;	(*Abfrage Istdrehzahl = 0*)		
	Q_bUmrDrehzNnenn	:BOOL;	(*Abfrage Drehzahl = Sollwert*)
	
	Q_stSEWOutput		:ST_SEWOutput;	(*SEW-Ausgänge*)

	Q_bAnstNetzUmr		:BOOL;	(*Netzansteuerung Umrichter*)
	Q_bAnstReglFrg		:BOOL;	(*Reglerfreigabe Umrichter*)

END_VAR
VAR CONSTANT
																					
	cSEW_Skalierg		:LREAL:= 16384;	(*16384 entspricht 100%*)

END_VAR
VAR
																						
	rtrigHandFkt0		:R_TRIG;													
	rtrigHandFkt1		:R_TRIG;									
																						{attribute 'hide'}
	bHdFktReset			:BOOL;
																						{attribute 'hide'}
	bEndstFrg			:BOOL;													{attribute 'hide'}
	bUmrStat				:BOOL;													{attribute 'hide'}
	bDatenFrg			:BOOL;													{attribute 'hide'}
	bUmrFehl				:BOOL;													{attribute 'hide'}
	nIstDrehz			:INT;														{attribute 'hide'}
	nIstStrom			:INT;
																						{attribute 'hide'}
	bReglSperr			:BOOL;													{attribute 'hide'}
	bSchnStop			:BOOL;													{attribute 'hide'}
	bDrehzFrg			:BOOL;													{attribute 'hide'}
	bUmrReset			:BOOL;													{attribute 'hide'}
	nSollDrehz			:INT;														{attribute 'hide'}
	fSollRamp			:WORD;
																						{attribute 'hide'}
	tonDrehzNnull		:TON;														{attribute 'hide'}
	tonDrehzNnenn		:TON;
	
	tonMeldLaufzeit0	:TON;
	tonMeldLaufzeit1	:TON;
	
	tonMeldNichtBtb				: TON; 	// Meldeverzögerung für Nicht BTB, da der Umrichterstatus erst verzögert kommt
	tonMeldUmrichterGesperrt	: TON;	// Meldeverzögerung für "Umrichter gesperrt"-Meldung. Das Bit bEndstFrg kommt erst ca 22ms nach der Freigabe
	
	//Relevante Variablen zur Diagnose
	stUniAnstgFkt		:ST_UniBaustein;

	//Zus. Variablen Betrieb HF-Aggregate
	nStepEinlZykl		:INT;
	nEinlZyklPhase		:INT;
	tonEinlZyklPhase	:TON;
	arrEinlZyklPhase	:ARRAY[1..21] OF TIME := [T#1M, T#2M, T#1M, T#2M, T#1M, T#2M, T#1M, T#2M, T#1M, T#2M, T#1M, T#2M, T#1M, T#2M, T#1M, T#2M, T#30M, T#5M, T#30M, T#5M];
	arrEinlZyklDrehz	:ARRAY[1..21] OF LREAL:= [33, 0, 33, 0, 33, 0, 66, 0, 66, 0, 66, 0, 100, 0, 100, 0, 100, 0, 100, 0];
	nDrehzEinlZykl		:LREAL;

	nStepBetrZykl		:INT;
	nBetrZyklPhase		:INT;
	tonBetrZyklPhase	:TON;
	nDrehzBetrZykl		:LREAL;

	bHochlZyklStart	:BOOL;	
	bHochlZyklEnde		:BOOL;
	
	nAktlSollwVorg		:LREAL;
	
	nFehlercode				: DWORD;
	sFehlerstring			: STRING;
	sLetzerFehlerstring	: STRING;
	tonVerzFehlerstring	: TON;
	
	bUmrichterGesperrt	: BOOL;
	
END_VAR

	(*Uni.- Antriebsansteuerung /SEW-Umrichter(EtherCAT)*)
	
	(**************************************************)	
	(*Aufruf-Bereichskontrolle*)

	IF I_nSchutzBer <= 0 OR I_nSchutzBer > cAnzSchutzBer
		OR ((NOT __ISVALIDREF(I_RefAchse)
				OR NOT __ISVALIDREF(I_RefAxis))
			AND I_eAntriebTyp = E_AntriebTyp.eEilSchleich)
		OR	I_nAntrEinsGrp <= 0 OR I_nAntrEinsGrp > cAnzEinschGrp
		OR I_fSollwMaxUmr <= 0
		// OR I_fSollwVrgUmr <= 0	// Sollwert darf 0 annehmen.
	THEN
		IF I_nSchutzBer <= 0 OR I_nSchutzBer > cAnzSchutzBer
		THEN
			IQ_stUniAnstgHMI.stMeldAusgHMI.sMeldText		:= 'I_nSchutzBer = 0 oder zu gross.';
		ELSIF I_nAntrEinsGrp <= 0 OR I_nAntrEinsGrp > cAnzEinschGrp
		THEN
			IQ_stUniAnstgHMI.stMeldAusgHMI.sMeldText		:= 'I_nAntrEinsGrp = 0 oder zu gross.';
		ELSIF I_fSollwMaxUmr <= 0
		THEN
			IQ_stUniAnstgHMI.stMeldAusgHMI.sMeldText		:= 'I_fSollwMaxUmr = 0 oder kleiner und IQ_stUniAnstgHMI.fVmax = 0 oder kleiner.';
		//ELSIF I_fSollwVrgUmr <= 0
		//THEN
		//	IQ_stUniAnstgHMI.stMeldAusgHMI.sMeldText		:= 'I_fSollwVrgUmr = 0 oder kleiner.';
		ELSE
			IQ_stUniAnstgHMI.stMeldAusgHMI.sMeldText		:= 'I_RefAchse oder I_RefAxis nicht beschrieben.';
		END_IF

		IQ_stUniAnstgHMI.stMeldAusgHMI.SourceName			:= I_sStatName;
		IQ_stUniAnstgHMI.stMeldAusgHMI.sAktorName			:= I_sAktorName;
		
		IF I_sAktorBMK <> ''
		THEN
			IQ_stUniAnstgHMI.stMeldAusgHMI.sBMK	:= I_sAktorBMK;
		ELSE
			IQ_stUniAnstgHMI.stMeldAusgHMI.sBMK	:= I_stVarInfoBMK.Comment;
		END_IF
		
		IQ_stUniAnstgHMI.stMeldAusgHMI.bMeldHinweis		:= bMaschParamAllgGueltig;
		
		// Texte der Handfunktionen zuweisen. Das sieht sonst schieße aus in der HMI
		stUniAnstgFkt.nHandStat	:= 256;	// Funktion sperren
		y_ZustAnzg();
		
		RETURN;
	ELSE
		IQ_stUniAnstgHMI.stMeldAusgHMI.bMeldHinweis	:= FALSE;
		IQ_stUniAnstgHMI.stMeldAusgHMI.sMeldText		:= '';
	END_IF

	(**************************************************)	
	(*Haendling Uni-Struktur*)

	CASE I_eAntriebTyp OF
		 
1:	(*Antriebstyp Aggregat*)
	
	a_Aggregat();

2:	(*Antriebstyp Transport*) 
	
	b_Transport();

3:	(*Antriebstyp Verstellg.*)

	c_Verstellg();	

4: (*Antriebstyp EilSchleich*)	
	
	d_EilSchleich();
	
5:	(*Antriebstyp HF-Aggregat*)
	
	a_Aggregat();

	u_AggEinlZykl(); //Einlaufphasen HF-Aggregat 
	v_AggBetrZykl(); //Betriebphasen HF-Aggregat
	
   END_CASE
	
	(**************************************************)	
	(*EtherCAT-Anschaltung*)	

	w_InOutSEW();

	(**************************************************)	
	(*Ausgänge zuweisen*)

	x_AusgZuw();
	
	(**************************************************)	
	(*Zustände anzeigen*)

	y_ZustAnzg();

	(**************************************************)	
	(*Meldungen ausgeben*)
	z_FehlerAusw();
	z_FehlMeld();
	
	(**************************************************)

ACTION a_Aggregat:
	(*Antriebstyp "Aggregat" /z.B. FU-Bohr.-Fräsaggregate...*)

	(*Verwendete Softkeytasten = 5 (s.Beispiel)*)

   (*       "Handfunktion"       /   "Softkeytaste 1"   /   "Softkeytaste 2"   /   "Softkeytaste 3"   /   "Softkeytaste 4"   /   "Softkeytaste 5"   *)
	(*                                                                          															  								 *) 
   (*------- Bohraggregat -------/_____ausschalten______/_____einschalten______/_________Frei_________/_________Frei_________/________Reset_________*)

	(*Softkeyleiste.1		:Funktion ausschalten	 *)
	(*Softkeyleiste.2		:Funktion einschalten	 *)
	(*Softkeyleiste.3		:Platzhalter				 *)
	(*Softkeyleiste.4		:Platzhalter				 *)
	(*Softkeyleiste.5		:Funktion Umrichter-Reset*)

	(*Hinweis:
	- Funktion wird durch "ResHdBetr" bei Betriebsartenwechsel zurückgenommen
	*)

	(**************************************************)	

	stUniAnstgFkt.bHandAnw0:= IQ_stUniAnstgHMI.stHandFktHMI[1].bySwitch > 0;
	stUniAnstgFkt.bHandAnw1:= IQ_stUniAnstgHMI.stHandFktHMI[2].bySwitch > 0;

	bHdFktReset				  := IQ_stUniAnstgHMI.stHandFktHMI[5].bySwitch > 0;	
	
	IF arrBetrartAutomAktiv[I_nSchutzBer]
		OR I_bResHandFkt
		OR bHdFktReset
		OR NOT I_bExtReglFrg
		OR NOT arrAntrGruppeFrg[I_nSchutzBer]
		THEN
			stUniAnstgFkt.arrHandFkt[1]:= FALSE;
		ELSE
			IF arrBetrartAutomSpeichn[I_nSchutzBer]
				THEN
					IF NOT I_bResHdBetr THEN
						stUniAnstgFkt.arrHandFkt[1]:= stUniAnstgFkt.arrFktAusfg[1];
					END_IF
				ELSE
					IF NOT arrGrdstlgBetrAktiv[I_nSchutzBer]
						AND arrBetrartHandAktiv[I_nSchutzBer]
						THEN
							 IF stUniAnstgFkt.bHandAnw1 THEN
								 stUniAnstgFkt.arrHandFkt[1]:= TRUE;
							 END_IF
							 IF stUniAnstgFkt.bHandAnw0 THEN
								 stUniAnstgFkt.arrHandFkt[1]:= FALSE;
							 END_IF
					END_IF
			END_IF
	END_IF

	IF arrBetrartHandAktiv[I_nSchutzBer]
		THEN
			IF stUniAnstgFkt.arrHandFkt[1]
				THEN
					stUniAnstgFkt.nHandStat:= 2;	(*Handfunktion.2 aktiv*)
				ELSE
					stUniAnstgFkt.nHandStat:= 1;	(*Handfunktion.1 aktiv*)
			END_IF
		ELSE
			stUniAnstgFkt.nHandStat:= 256;		(*Funktion gesperrt*)
	END_IF

	(**************************************************)	

	IF arrBetrartHandAktiv[I_nSchutzBer]
		THEN
			stUniAnstgFkt.arrGrdstFkt[1]:= I_arrZuwGrdstFkt[1];
		ELSE
			stUniAnstgFkt.arrGrdstFkt[1]:= FALSE;
   END_IF
	IF arrBetrartAutomAktiv[I_nSchutzBer] OR TRUE //ToDo
		THEN
			stUniAnstgFkt.arrAutomFkt[1]:= I_arrZuwAutomFkt[1];
		ELSE
			stUniAnstgFkt.arrAutomFkt[1]:= FALSE;
   END_IF

	(**************************************************)	

	stUniAnstgFkt.arrFktAusfg[1]:= stUniAnstgFkt.arrGrdstFkt[1]
										 	 OR stUniAnstgFkt.arrHandFkt[1]
										 	 OR stUniAnstgFkt.arrAutomFkt[1];

	(**************************************************)
END_ACTION

ACTION b_Transport:
	(*Antriebstyp "Transport" /z.B. FU-Transportsegmente...*)

	(*Verwendete Softkeytasten = 5 (s.Beispiel)*)

   (*       "Handfunktion"       /   "Softkeytaste 1"   /   "Softkeytaste 2"   /   "Softkeytaste 3"   /   "Softkeytaste 4"   /   "Softkeytaste 5"   *)
	(*                                                                          															  								 *) 
	(*----- Transportantrieb -----/_einschalten (zurück)_/___einschalten (vor)__/_______langsam________/_______schnell________/________Reset_________*)

	(*Softkeyleiste.1		:Funktion ein.-ausschalten Reversierend*)
	(*Softkeyleiste.2		:Funktion ein.-ausschalten             *)
	(*Softkeyleiste.3		:Funktion langsame Drehzahl (SollwMin) *)
	(*Softkeyleiste.4		:Funktion schnelle Drehzahl (SollwVrg) *)
	(*Softkeyleiste.5		:Funktion Umrichter-Reset				   *)

	(*Hinweis:
	- Funktion wird durch "VerrHdFkt" gesperrt (z.B. kein Reversierbetrieb...)
	*)

	(**************************************************)	

	stUniAnstgFkt.bHandAnw0:= IQ_stUniAnstgHMI.stHandFktHMI[1].bySwitch > 0;
	stUniAnstgFkt.bHandAnw1:= IQ_stUniAnstgHMI.stHandFktHMI[2].bySwitch > 0;
	stUniAnstgFkt.bHandAnw2:= IQ_stUniAnstgHMI.stHandFktHMI[3].bySwitch > 0;
	stUniAnstgFkt.bHandAnw3:= IQ_stUniAnstgHMI.stHandFktHMI[4].bySwitch > 0;
	bHdFktReset				  := IQ_stUniAnstgHMI.stHandFktHMI[5].bySwitch > 0;	
	
	IF arrBetrartAutomAktiv[I_nSchutzBer]
		OR I_bResHandFkt
		OR bHdFktReset
		OR NOT I_bExtReglFrg
		THEN
			stUniAnstgFkt.arrHandFkt[0]:=
			stUniAnstgFkt.arrHandFkt[1]:=
			stUniAnstgFkt.arrHandFkt[2]:=
			stUniAnstgFkt.arrHandFkt[3]:= FALSE;
		ELSE
			IF NOT arrBetrartAutomSpeichn[I_nSchutzBer]
				THEN
					IF NOT arrGrdstlgBetrAktiv[I_nSchutzBer]
						THEN
							 rtrigHandFkt1 (CLK:= stUniAnstgFkt.bHandAnw1);
							 IF rtrigHandFkt1.Q THEN
								 stUniAnstgFkt.arrHandFkt[1]:= NOT stUniAnstgFkt.arrHandFkt[1];
							 END_IF
							 IF NOT arrBetrartHandAktiv[I_nSchutzBer]
								 OR stUniAnstgFkt.arrHandFkt[0]
								 OR I_bVerrHdFktV THEN
								 stUniAnstgFkt.arrHandFkt[1]:= FALSE;
							 END_IF
	 
							 rtrigHandFkt0 (CLK:= stUniAnstgFkt.bHandAnw0);
							 IF rtrigHandFkt0.Q THEN
								 stUniAnstgFkt.arrHandFkt[0]:= NOT stUniAnstgFkt.arrHandFkt[0];
							 END_IF
							 IF NOT arrBetrartHandAktiv[I_nSchutzBer]
								 OR stUniAnstgFkt.arrHandFkt[1]
								 OR I_bVerrHdFktZ THEN
								 stUniAnstgFkt.arrHandFkt[0]:= FALSE;
							 END_IF
	 
							 IF stUniAnstgFkt.bHandAnw3 THEN
								 stUniAnstgFkt.arrHandFkt[3]:= TRUE;
							 END_IF
							 IF NOT arrBetrartHandAktiv[I_nSchutzBer]
								 OR stUniAnstgFkt.bHandAnw2 THEN
								 stUniAnstgFkt.arrHandFkt[3]:= FALSE;
							 END_IF
					END_IF
			END_IF
	END_IF

	IF arrBetrartHandAktiv[I_nSchutzBer]
		THEN
			stUniAnstgFkt.nHandStat:= 0;			(*Funktion freigegeben*)
			IF stUniAnstgFkt.arrHandFkt[1]
				THEN
					stUniAnstgFkt.nHandStat:= 2;	(*Handfunktion.2 aktiv*)
			END_IF
			IF stUniAnstgFkt.arrHandFkt[0]
				THEN
					stUniAnstgFkt.nHandStat:= 1;	(*Handfunktion.1 aktiv*)
			END_IF
			IF stUniAnstgFkt.arrHandFkt[3]
				THEN
					stUniAnstgFkt.nHandStat:=
					stUniAnstgFkt.nHandStat + 8;	(*Handfunktion.4 aktiv*)
				ELSE
					stUniAnstgFkt.nHandStat:=
					stUniAnstgFkt.nHandStat + 4;	(*Handfunktion.3 aktiv*)
			END_IF
		ELSE
			stUniAnstgFkt.nHandStat:= 256;		(*Funktion gesperrt*)
	END_IF

	(**************************************************)	

	IF arrBetrartHandAktiv[I_nSchutzBer]
		THEN
			stUniAnstgFkt.arrGrdstFkt[0]:= I_arrZuwGrdstFkt[0];
			stUniAnstgFkt.arrGrdstFkt[1]:= I_arrZuwGrdstFkt[1];
			stUniAnstgFkt.arrGrdstFkt[3]:= I_arrZuwGrdstFkt[2];
		ELSE
			stUniAnstgFkt.arrGrdstFkt[0]:= 
			stUniAnstgFkt.arrGrdstFkt[1]:=
			stUniAnstgFkt.arrGrdstFkt[3]:= FALSE;
   END_IF
	IF arrBetrartAutomAktiv[I_nSchutzBer] OR TRUE //ToDo
		THEN
			stUniAnstgFkt.arrAutomFkt[0]:= I_arrZuwAutomFkt[0];
			stUniAnstgFkt.arrAutomFkt[1]:= I_arrZuwAutomFkt[1];
			stUniAnstgFkt.arrAutomFkt[3]:= I_arrZuwAutomFkt[2];
		ELSE
			stUniAnstgFkt.arrAutomFkt[0]:= 
			stUniAnstgFkt.arrAutomFkt[1]:= 
			stUniAnstgFkt.arrAutomFkt[3]:= FALSE;
   END_IF

	(**************************************************)	

	stUniAnstgFkt.arrFktAusfg[0]:= stUniAnstgFkt.arrGrdstFkt[0]
										 	 OR stUniAnstgFkt.arrHandFkt[0]
										 	 OR stUniAnstgFkt.arrAutomFkt[0];

	stUniAnstgFkt.arrFktAusfg[1]:= stUniAnstgFkt.arrGrdstFkt[1]
										 	 OR stUniAnstgFkt.arrHandFkt[1]
										 	 OR stUniAnstgFkt.arrAutomFkt[1];

	stUniAnstgFkt.arrFktAusfg[3]:= stUniAnstgFkt.arrGrdstFkt[3]
										 	 OR stUniAnstgFkt.arrHandFkt[3]
										 	 OR stUniAnstgFkt.arrAutomFkt[3];

	(**************************************************)
END_ACTION

ACTION c_Verstellg:
	(*Antriebstyp "Verstellg." /z.B. FU-Antriebe mit Eil/Schleichbewegung...*)

	(*Verwendete Softkeytasten = 5 (s.Beispiel)*)

   (*       "Handfunktion"       /   "Softkeytaste 1"   /   "Softkeytaste 2"   /   "Softkeytaste 3"   /   "Softkeytaste 4"   /   "Softkeytaste 5"   *)
	(*                                                                          															  								 *) 
	(*----- Verstellantrieb ------/_____zurückfahren_____/_______vorfahren______/_______langsam________/_______schnell________/________Reset_________*)

	(*Softkeyleiste.1		:Funktion ein.-ausschalten Reversierend*)
	(*Softkeyleiste.2		:Funktion ein.-ausschalten             *)
	(*Softkeyleiste.3		:Funktion langsame Drehzahl (SollwMin) *)
	(*Softkeyleiste.4		:Funktion schnelle Drehzahl (SollwVrg) *)
	(*Softkeyleiste.5		:Funktion Umrichter-Reset				   *)

	(*Hinweis:
	- Funktion wird durch "VerrHdFkt" gesperrt (z.B. bei Überstandserkennung...)
	- Funktion wird durch "EndlHdFkt/VerzHdFkt" zurückgenommen bzw. umgeschaltet
	*)
	
	(**************************************************)	

	stUniAnstgFkt.bHandAnw0:= IQ_stUniAnstgHMI.stHandFktHMI[1].bySwitch > 0;
	stUniAnstgFkt.bHandAnw1:= IQ_stUniAnstgHMI.stHandFktHMI[2].bySwitch > 0;
	stUniAnstgFkt.bHandAnw2:= IQ_stUniAnstgHMI.stHandFktHMI[3].bySwitch > 0;
	stUniAnstgFkt.bHandAnw3:= IQ_stUniAnstgHMI.stHandFktHMI[4].bySwitch > 0;
	bHdFktReset				  := IQ_stUniAnstgHMI.stHandFktHMI[5].bySwitch > 0;	
	
	IF arrBetrartAutomAktiv[I_nSchutzBer]
		OR I_bResHandFkt
		OR bHdFktReset
		OR NOT I_bExtReglFrg
		THEN
			stUniAnstgFkt.arrHandFkt[0]:=
			stUniAnstgFkt.arrHandFkt[1]:=
			stUniAnstgFkt.arrHandFkt[2]:=
			stUniAnstgFkt.arrHandFkt[3]:= FALSE;
		ELSE
			IF NOT arrBetrartAutomSpeichn[I_nSchutzBer]
				THEN
					IF NOT arrGrdstlgBetrAktiv[I_nSchutzBer]
						THEN
							 rtrigHandFkt1 (CLK:= stUniAnstgFkt.bHandAnw1);
							 IF rtrigHandFkt1.Q THEN
								 stUniAnstgFkt.arrHandFkt[1]:= NOT stUniAnstgFkt.arrHandFkt[1];
							 END_IF
							 IF NOT arrBetrartHandAktiv[I_nSchutzBer]
								 OR stUniAnstgFkt.arrHandFkt[0]
								 OR I_bVerrHdFktV OR NOT I_bEndlHdFktV THEN
								 stUniAnstgFkt.arrHandFkt[1]:= FALSE;
							 END_IF
	 
							 rtrigHandFkt0 (CLK:= stUniAnstgFkt.bHandAnw0);
							 IF rtrigHandFkt0.Q THEN
								 stUniAnstgFkt.arrHandFkt[0]:= NOT stUniAnstgFkt.arrHandFkt[0];
							 END_IF
							 IF NOT arrBetrartHandAktiv[I_nSchutzBer]
								 OR stUniAnstgFkt.arrHandFkt[1]
								 OR I_bVerrHdFktZ OR NOT I_bEndlHdFktZ THEN
								 stUniAnstgFkt.arrHandFkt[0]:= FALSE;
							 END_IF
	 
							 IF stUniAnstgFkt.bHandAnw3 THEN
								 stUniAnstgFkt.arrHandFkt[3]:= TRUE;
							 END_IF
							 IF NOT arrBetrartHandAktiv[I_nSchutzBer]
								 OR (stUniAnstgFkt.arrHandFkt[1] AND I_bVerzHdFktV)
								 OR (stUniAnstgFkt.arrHandFkt[0] AND I_bVerzHdFktZ)
								 OR stUniAnstgFkt.bHandAnw2 THEN
								 stUniAnstgFkt.arrHandFkt[3]:= FALSE;
							 END_IF
					END_IF
			END_IF
	END_IF

	IF arrBetrartHandAktiv[I_nSchutzBer]
		THEN
			stUniAnstgFkt.nHandStat:= 0;			(*Funktion freigegeben*)
			IF stUniAnstgFkt.arrHandFkt[1]
				THEN
					stUniAnstgFkt.nHandStat:= 2;	(*Handfunktion.2 aktiv*)
			END_IF
			IF stUniAnstgFkt.arrHandFkt[0]
				THEN
					stUniAnstgFkt.nHandStat:= 1;	(*Handfunktion.1 aktiv*)
			END_IF
			IF stUniAnstgFkt.arrHandFkt[3]
				THEN
					stUniAnstgFkt.nHandStat:=
					stUniAnstgFkt.nHandStat + 8;	(*Handfunktion.4 aktiv*)
				ELSE
					stUniAnstgFkt.nHandStat:=
					stUniAnstgFkt.nHandStat + 4;	(*Handfunktion.3 aktiv*)
			END_IF
		ELSE
			stUniAnstgFkt.nHandStat:= 256;		(*Funktion gesperrt*)
	END_IF

	(**************************************************)	

	IF arrBetrartHandAktiv[I_nSchutzBer]
		THEN
			stUniAnstgFkt.arrGrdstFkt[0]:= I_arrZuwGrdstFkt[0];
			stUniAnstgFkt.arrGrdstFkt[1]:= I_arrZuwGrdstFkt[1];
			stUniAnstgFkt.arrGrdstFkt[3]:= I_arrZuwGrdstFkt[2];
		ELSE
			stUniAnstgFkt.arrGrdstFkt[0]:= 
			stUniAnstgFkt.arrGrdstFkt[1]:=
			stUniAnstgFkt.arrGrdstFkt[3]:= FALSE;
   END_IF
	IF arrBetrartAutomAktiv[I_nSchutzBer] OR TRUE //ToDo
		THEN
			stUniAnstgFkt.arrAutomFkt[0]:= I_arrZuwAutomFkt[0];
			stUniAnstgFkt.arrAutomFkt[1]:= I_arrZuwAutomFkt[1];
			stUniAnstgFkt.arrAutomFkt[3]:= I_arrZuwAutomFkt[2];
		ELSE
			stUniAnstgFkt.arrAutomFkt[0]:= 
			stUniAnstgFkt.arrAutomFkt[1]:= 
			stUniAnstgFkt.arrAutomFkt[3]:= FALSE;
   END_IF

	(**************************************************)	

	stUniAnstgFkt.arrFktAusfg[0]:= (stUniAnstgFkt.arrGrdstFkt[0]
										 	 	OR stUniAnstgFkt.arrHandFkt[0]
										 	 	OR stUniAnstgFkt.arrAutomFkt[0])
											AND I_bEndlHdFktZ;

	stUniAnstgFkt.arrFktAusfg[1]:= (stUniAnstgFkt.arrGrdstFkt[1]
										 	 OR stUniAnstgFkt.arrHandFkt[1]
										 	 OR stUniAnstgFkt.arrAutomFkt[1])
											AND I_bEndlHdFktV;

	stUniAnstgFkt.arrFktAusfg[3]:= (stUniAnstgFkt.arrGrdstFkt[3]
												 OR stUniAnstgFkt.arrHandFkt[3]
												 OR stUniAnstgFkt.arrAutomFkt[3])
											AND(( stUniAnstgFkt.arrFktAusfg[0]
													AND NOT I_bVerzHdFktZ)
												OR ( stUniAnstgFkt.arrFktAusfg[1]
													AND NOT I_bVerzHdFktV));

	(**************************************************)
END_ACTION

ACTION d_EilSchleich:
	(*Antriebstyp "EilSchleich" /z.B. FU-Antriebe mit Eil/Schleichachse...*)

	(*Verwendete Softkeytasten = 5 (s.Beispiel)*)

   (*       "Handfunktion"       /   "Softkeytaste 1"   /   "Softkeytaste 2"   /   "Softkeytaste 3"   /   "Softkeytaste 4"   /   "Softkeytaste 5"   *)
	(*                                                                          															  								 *) 
	(*------ Verstellachse -------/____negativ fahren____/____positiv fahren____/_________Frei_________/_________Frei_________/________Reset_________*)
	
	(*Softkeyleiste.1		:Funktion Tastend aktiv /Richtg. Negativ*)
	(*Softkeyleiste.2		:Funktion Tastend aktiv /Richtg. Positiv*)
	(*Softkeyleiste.3		:Platzhalter				 					 *)
	(*Softkeyleiste.4		:Platzhalter				 					 *)
	(*Softkeyleiste.5		:Funktion Umrichter-Reset					 *)

	(*Hinweis:
	- Funktion wird durch "VerrHdFkt" gesperrt (z.B. bei Überstandserkennung...)
	*)

	(**************************************************)	

	stUniAnstgFkt.bHandAnw0:= IQ_stUniAnstgHMI.stHandFktHMI[1].bySwitch > 0;
	stUniAnstgFkt.bHandAnw1:= IQ_stUniAnstgHMI.stHandFktHMI[2].bySwitch > 0;
	bHdFktReset				  := IQ_stUniAnstgHMI.stHandFktHMI[5].bySwitch > 0;	
	
	IF arrBetrartAutomAktiv[I_nSchutzBer]
		OR bHdFktReset
		OR NOT I_bExtReglFrg
		THEN
			stUniAnstgFkt.arrHandFkt[0]:=
			stUniAnstgFkt.arrHandFkt[1]:= FALSE;
		ELSE
			IF NOT arrBetrartAutomSpeichn[I_nSchutzBer] THEN
				IF NOT arrGrdstlgBetrAktiv[I_nSchutzBer] THEN
					stUniAnstgFkt.arrHandFkt[1]:= arrBetrartHandAktiv[I_nSchutzBer]
													  		AND stUniAnstgFkt.bHandAnw1
													  		AND NOT stUniAnstgFkt.bHandAnw0
													  		AND NOT I_bVerrHdFktV	
													  		AND I_RefAchse.stFreigb.bVorsFrgPos;
					stUniAnstgFkt.arrHandFkt[0]:= arrBetrartHandAktiv[I_nSchutzBer]
													  		AND stUniAnstgFkt.bHandAnw0
													  		AND NOT stUniAnstgFkt.bHandAnw1
													  		AND NOT I_bVerrHdFktZ
													  		AND I_RefAchse.stFreigb.bVorsFrgNeg;
				END_IF
			END_IF
	END_IF

	IF arrBetrartHandAktiv[I_nSchutzBer]
		THEN
			stUniAnstgFkt.nHandStat:= 0;			(*Funktion freigegeben*)
			IF stUniAnstgFkt.arrHandFkt[1]
				THEN
					stUniAnstgFkt.nHandStat:= 2;	(*Handfunktion.2 aktiv*)
			END_IF
			IF stUniAnstgFkt.arrHandFkt[0]
				THEN
					stUniAnstgFkt.nHandStat:= 1;	(*Handfunktion.1 aktiv*)
			END_IF
		ELSE
			stUniAnstgFkt.nHandStat:= 256;		(*Funktion gesperrt*)
	END_IF

	(**************************************************)	
	
	I_RefAchse.stStatus.bAchseBTB	:= Q_bAbfrStatUmr;

	I_RefAchse.stGrdfkt.bHdfkt_pos:=	stUniAnstgFkt.arrHandFkt[1];
	I_RefAchse.stGrdfkt.bHdfkt_neg:=	stUniAnstgFkt.arrHandFkt[0];

	(**************************************************)
END_ACTION

ACTION u_AggEinlZykl:
	(*Inbetriebnahme HF-Aggregate (Einlaufphasen f. optimale Fettverteilung)*)

	nAktlSollwVorg	:= 0; //Init.

	IF NOT I_bAnwEinlZykl
		OR arrTaktStopWartungsTuer[I_nSchutzBer]
	THEN
		nStepEinlZykl	:= 0;		 

		RETURN;
	END_IF

	(**************************************************)	

CASE nStepEinlZykl OF
0:
	//Initialisierung:
	nDrehzEinlZykl	:= 0;
	
	tonEinlZyklPhase (IN:= FALSE);
	nEinlZyklPhase	:= 1;

	IF stUniAnstgFkt.arrHandFkt[1] THEN
		nStepEinlZykl:= 100;
   END_IF

100, 110, 120, 130, 140, 150, 160, 170, 180, 190, 200, 210, 220, 230, 240, 250, 260, 270, 280, 290:
	//Einlaufphasen 1-20:

	nDrehzEinlZykl:= (I_fSollwMaxUmr * (arrEinlZyklDrehz[nEinlZyklPhase] / 100));
	
	tonEinlZyklPhase (IN:= stUniAnstgFkt.arrHandFkt[1],
							PT:= arrEinlZyklPhase[nEinlZyklPhase]);
	
	IF tonEinlZyklPhase.Q THEN
		tonEinlZyklPhase (IN:= FALSE);
		nEinlZyklPhase:= nEinlZyklPhase + 1;
		
		nStepEinlZykl:= nStepEinlZykl + 10;		 
	END_IF	

	IF NOT stUniAnstgFkt.arrHandFkt[1] THEN
		nStepEinlZykl:= 0;		 
   END_IF
	
300:
	//Ende Einlaufzyklus
	nStepEinlZykl:= nStepEinlZykl;		 
	
END_CASE

	nAktlSollwVorg:= nDrehzEinlZykl;
	
	(**************************************************)
END_ACTION

ACTION v_AggBetrZykl:
	(*Betriebszyklen HF-Aggregate (Warmlaufphasen z. Verschleißminderung)*)

	IF I_bAnwEinlZykl THEN
		nStepBetrZykl	:= 0;		 
		bHochlZyklStart:=
		bHochlZyklEnde	:= FALSE;

		RETURN;
	END_IF

	(**************************************************)	

	IF (stUniAnstgFkt.arrFktAusfg[1]	//Optional weitere Bedingungen? 
			OR I_bStandbyBetr)
		AND arrBetrartAutomAktiv[I_nSchutzBer]
		THEN //Betriebszyklus start
			bHochlZyklStart:= TRUE;	

	ELSIF FALSE (*Optional*)
		THEN //Betriebszyklus stop
			bHochlZyklStart:= FALSE;	

			nStepBetrZykl:= 0;		 

	ELSIF NOT stUniAnstgFkt.arrFktAusfg[1]
		 	AND NOT I_bStandbyBetr
		THEN //Betriebszyklus halt 
			bHochlZyklStart:= FALSE;	

	END_IF

	(**************************************************)	
	
CASE nStepBetrZykl OF
0:
	//Initialisierung:
	nDrehzBetrZykl:= 0;

	bHochlZyklEnde:= FALSE;	
	
	tonBetrZyklPhase (IN:= FALSE);
	nBetrZyklPhase:= 0;
	
	IF bHochlZyklStart THEN
		nStepBetrZykl:= 100;		 
   END_IF

100, 200, 300:
	//Hochlaufphasen 1-3:
	nBetrZyklPhase:= nStepBetrZykl / 100; 

	nDrehzBetrZykl:= (I_fSollwMaxUmr * (I_arrBetrZyklDrehz[nBetrZyklPhase] / 100));

	tonBetrZyklPhase (IN:= bHochlZyklStart,
							PT:= I_arrBetrZyklPhase[nBetrZyklPhase]);
	
	IF NOT arrBetrartAutomAktiv[I_nSchutzBer]
	THEN	// Hochlaufzyklus unterbrechen, wenn Schutztür angewählt wurde
		bHochlZyklStart	:= FALSE;
	END_IF

	IF tonBetrZyklPhase.Q THEN
		tonBetrZyklPhase (IN:= FALSE);
		
		nStepBetrZykl:= nStepBetrZykl + 100;		 

	ELSIF NOT bHochlZyklStart THEN
		tonBetrZyklPhase (IN:= FALSE);
		
		nStepBetrZykl:= nStepBetrZykl * -1;		 
	END_IF	

400:
	//Ende Hochlaufzyklus => Betriebsbereit
	nBetrZyklPhase	:= nStepBetrZykl / 100; 

	bHochlZyklEnde	:= TRUE;
	
	IF stUniAnstgFkt.arrFktAusfg[1]
	THEN	//Bearbeitungsdrehzahl
		nDrehzBetrZykl	:= I_fSollwVrgUmr;
		
	ELSIF NOT arrBetrartAutomAktiv[I_nSchutzBer]
		OR arrAutoStopWartungsTuer[I_nSchutzBer]
	THEN	// wenn Automatik ausgeht, z.B. bei Schutztüranwahl, dann soll der Motor stehen. Aber nur wenn nicht noch stUniAnstgFkt.arrFktAusfg[1] ansteht.
		nDrehzBetrZykl	:= 0;

	ELSE	//Leerlaufdrehzahl
		nDrehzBetrZykl	:= (I_fSollwMaxUmr * (I_arrBetrZyklDrehz[nBetrZyklPhase] / 100));
		
   END_IF

	tonBetrZyklPhase (IN:= NOT bHochlZyklStart,
							PT:= I_arrBetrZyklPhase[nBetrZyklPhase]);
	
	IF tonBetrZyklPhase.Q THEN
		tonBetrZyklPhase (IN:= FALSE);

		bHochlZyklEnde	:= FALSE;
		
		nStepBetrZykl	:= 500;		 
	END_IF

500:
	//Stillstandphase > 15min
	tonBetrZyklPhase (IN:= TRUE,
							PT:= I_tPause);
	
	IF tonBetrZyklPhase.Q THEN
		tonBetrZyklPhase (IN:= FALSE);
	
		nStepBetrZykl:= 0;		 

	ELSIF bHochlZyklStart THEN 
		tonBetrZyklPhase (IN:= FALSE);

		IF tonBetrZyklPhase.ET > (I_tPause/2) //Halbe Stillstandszeit
			THEN		
				nStepBetrZykl:= 300; //Erneuter Hochlauf ab Phase 3 			 
			ELSE
				nStepBetrZykl:= 400; //Direkt wieder Betriebsbereit		 
	  END_IF
	END_IF	
	
	nDrehzBetrZykl:= 0;

ELSE	// Hier wird reingesprungen, wenn die Schritte negativ werden.
	
	//Hochlaufphase Unterbrochen 
	tonBetrZyklPhase (IN:= TRUE,
							PT:= T#15S);
							
	nDrehzBetrZykl	:= 0;	// Wenn die Hochlaufphase unterbrochen wurde, die Drehzahl auf 0 setzen
	
	IF tonBetrZyklPhase.Q THEN
		tonBetrZyklPhase (IN:= FALSE);

		CASE nStepBetrZykl OF
		-100:	nStepBetrZykl:= 0;	
		-200:	nStepBetrZykl:= 100;	
		-300:	nStepBetrZykl:= 200;	
	  	END_CASE

	ELSIF bHochlZyklStart THEN 
		tonBetrZyklPhase (IN:= FALSE);

		nStepBetrZykl:= nStepBetrZykl * -1;		 

	END_IF	

END_CASE

	nAktlSollwVorg:= nDrehzBetrZykl;
	
	(**************************************************)
END_ACTION

ACTION w_InOutSEW:

	(**************************************************)	
	(*EtherCAT-Anschaltung*)	

	bEndstFrg:= I_stSEWInput.arrPI[1].0;
	bUmrStat	:= I_stSEWInput.arrPI[1].1;
	bDatenFrg:= I_stSEWInput.arrPI[1].2;
	bUmrFehl	:= I_stSEWInput.arrPI[1].5;
	nFehlercode.0	:= I_stSEWInput.arrPI[1].8;
	nFehlercode.1	:= I_stSEWInput.arrPI[1].9;
	nFehlercode.2	:= I_stSEWInput.arrPI[1].10;
	nFehlercode.3	:= I_stSEWInput.arrPI[1].11;
	nFehlercode.4	:= I_stSEWInput.arrPI[1].12;
	nFehlercode.5	:= I_stSEWInput.arrPI[1].13;
	nFehlercode.6	:= I_stSEWInput.arrPI[1].14;
	nFehlercode.7	:= I_stSEWInput.arrPI[1].15;
	
	nIstDrehz:= TO_INT(I_stSEWInput.arrPI[2]);
	nIstStrom:= TO_INT(I_stSEWInput.arrPI[3]);
	

	(**)

	bReglSperr:= NOT arrAntrGruppeFrg[I_nSchutzBer]
					 OR NOT I_bExtReglFrg
					 OR NOT bUmrStat
					 OR NOT bDatenFrg;
	bSchnStop := TRUE;
	bUmrReset := (NOT arrAntrGruppeFrg[I_nSchutzBer]
					 OR I_bUmrReset
					 OR bHdFktReset)
				    AND bUmrFehl;

	IF I_eAntriebTyp = 1 (*Typ Aggregat*)
		THEN
			IF stUniAnstgFkt.arrFktAusfg[1] 
				THEN
					nSollDrehz:= TO_INT(cSEW_Skalierg * LIMIT(I_fSollwMinUmr, I_fSollwVrgUmr, I_fSollwMaxUmr) / I_fSollwMaxUmr);

					bDrehzFrg := bUmrStat
								    AND bDatenFrg;
				ELSE
					nSollDrehz:= 0;
					bDrehzFrg := FALSE;
			END_IF
	ELSIF I_eAntriebTyp = 2 OR I_eAntriebTyp = 3 (*Typ Transport/Verstellg.*)
		THEN
			IF stUniAnstgFkt.arrFktAusfg[0] OR stUniAnstgFkt.arrFktAusfg[1] 
				THEN
					IF stUniAnstgFkt.arrFktAusfg[3]
						THEN
							nSollDrehz:= TO_INT(cSEW_Skalierg * LIMIT(I_fSollwMinUmr, I_fSollwVrgUmr, I_fSollwMaxUmr) / I_fSollwMaxUmr);
						ELSE
				 			nSollDrehz:= TO_INT(cSEW_Skalierg * I_fSollwMinUmr / I_fSollwMaxUmr);
					END_IF
					IF stUniAnstgFkt.arrFktAusfg[0]
						THEN
							nSollDrehz:= -(nSollDrehz);
					END_IF
					bDrehzFrg := bUmrStat
								    AND bDatenFrg;
				ELSE
					nSollDrehz:= 0;
					bDrehzFrg := FALSE;
			END_IF
	ELSIF I_eAntriebTyp = 4 (*Typ EilSchleich*)
		THEN
			IF (I_RefAxis.Status.PositiveDirection OR I_RefAxis.Status.NegativeDirection)
				AND I_RefAxis.NcToPlc.SetVelo > 0 
				THEN
					IF I_RefAxis.NcToPlc.SetVelo > 50
						AND I_RefAchse.stStatus.bInReferz
						THEN
							nSollDrehz:= TO_INT(cSEW_Skalierg * LIMIT(I_fSollwMinUmr, I_fSollwVrgUmr, I_fSollwMaxUmr) / I_fSollwMaxUmr);
						ELSE
				 			nSollDrehz:= TO_INT(cSEW_Skalierg * I_fSollwMinUmr / I_fSollwMaxUmr);
					END_IF
					IF I_RefAxis.Status.NegativeDirection
						THEN
							nSollDrehz:= -(nSollDrehz);
					END_IF
					bDrehzFrg := bUmrStat
								    AND bDatenFrg;
				ELSE
					nSollDrehz:= 0;
					bDrehzFrg := FALSE;
			END_IF
	ELSIF I_eAntriebTyp = 5 (*Typ Aggregat und HF-Betriebsart*)
		THEN
			IF nAktlSollwVorg > 0
				THEN
					nSollDrehz:= TO_INT(cSEW_Skalierg * LIMIT(0, nAktlSollwVorg, I_fSollwMaxUmr) / I_fSollwMaxUmr);
					
					bDrehzFrg := bUmrStat
								    AND bDatenFrg;
				ELSE
					nSollDrehz:= 0;
					bDrehzFrg := FALSE;
			END_IF
   END_IF

	// Drehzahl auf Maximum setzen
	IF bIbnMaxDrehz
	THEN
		nSollDrehz	:= TO_INT(cSEW_Skalierg);  
   END_IF
	
	IF NOT arrAntrGruppeFrg[I_nSchutzBer] (*Allg. Freigabe /..Fräser Abbremsen*)
	THEN		 
		nSollDrehz:= 0;
		bDrehzFrg := FALSE;
	END_IF

	IF ABS(nSollDrehz) > ABS(nIstDrehz)
	THEN
		fSollRamp:= TO_WORD(I_fRampVrgBUmr);
	ELSE
		fSollRamp:= TO_WORD(I_fRampVrgVUmr);
	END_IF
	
	(**)

	Q_bAbfrStatUmr		:= bUmrStat
								AND NOT IQ_stUniAnstgHMI.stMeldAusgHMI.bMeldUmrichterGesperrt;
								
	Q_nAbfrUmrDrehz	:= TO_INT((TO_LREAL(nIstDrehz) / cSEW_Skalierg) * 100);
	Q_nAbfrUmrStrom	:= (TO_INT(nIstStrom) / 10);

	Q_bUmrDrehzNnull	:=	Q_nAbfrUmrDrehz < 1;(*1%*)
	
	IF I_fSollwVrgUmr <> 0
	THEN	// Nur berechnen, wenn I_fSollwVrgUmr größer 0 ist, weil sonst durch 0 geteilt wird.
		Q_bUmrDrehzNnenn	:=	Q_nAbfrUmrDrehz > ((100 / (I_fSollwMaxUmr / I_fSollwVrgUmr)) * 0.95);(*95%*)
	ELSE	// Wenn I_fSollwVrgUmr = 0 Dann abfragen, ob Istdrehzahl 0 ist
		Q_bUmrDrehzNnenn	:= Q_nAbfrUmrDrehz < 1;
	END_IF

	tonDrehzNnull (IN:= Q_bUmrDrehzNnull,
						PT:= T#5S,//Filterzeit
						Q => Q_bUmrDrehzNnull);
	tonDrehzNnenn (IN:= Q_bUmrDrehzNnenn,
						PT:= T#5S,//Filterzeit
						Q => Q_bUmrDrehzNnenn);

	IF I_eAntriebTyp = 5
	THEN //Zus. Abfrage Hochlaufzyklus
		Q_bUmrDrehzNnenn	:=
			Q_bUmrDrehzNnenn
			AND bHochlZyklEnde; 
	END_IF

	(**)

	Q_stSEWOutput.arrPO[1].0:= bReglSperr;
	Q_stSEWOutput.arrPO[1].1:= bSchnStop;
	Q_stSEWOutput.arrPO[1].2:= bDrehzFrg;
	Q_stSEWOutput.arrPO[1].6:= bUmrReset;
	Q_stSEWOutput.arrPO[2]	:= TO_WORD(nSollDrehz);
	Q_stSEWOutput.arrPO[3]	:= fSollRamp;

	(**************************************************)
END_ACTION

ACTION x_AusgZuw:
	
	(**************************************************)	
	(*Ausgänge zuweisen*)
										
	CASE I_nAntrEinsGrp OF
1:	Q_bAnstNetzUmr:= arrAntrGruppe1Ein[I_nSchutzBer]
					  	  AND bVersEingAusgSchaltsOk;

2:	Q_bAnstNetzUmr:= arrAntrGruppe2Ein[I_nSchutzBer]
					  	  AND bVersEingAusgSchaltsOk;

3:	Q_bAnstNetzUmr:= arrAntrGruppe3Ein[I_nSchutzBer]
					  	  AND bVersEingAusgSchaltsOk;
	END_CASE

	Q_bAnstReglFrg:= arrAntrGruppeFrg[I_nSchutzBer]
						  AND I_bExtReglFrg
					  	  AND bUmrStat
					  	  AND bDatenFrg
					  	  AND bVersEingAusgSchaltsOk;

	(**************************************************)	
;
END_ACTION

ACTION y_ZustAnzg:
	
	(**************************************************)	
	(*Zustände anzeigen*)

	CASE I_eAntriebTyp OF
		 
1,5:(*Antriebstyp Aggregat*)
	
	IF stUniAnstgFkt.nHandStat = 1	(*Handfunktion.1 aktiv*)
		THEN
			IQ_stUniAnstgHMI.stHandFktHMI[1].sColour:= cGruenAsString; //eventl.: cRot;
			IQ_stUniAnstgHMI.stHandFktHMI[2].sColour:= cDefaultAsString;
			IQ_stUniAnstgHMI.stHandFktHMI[1].sText:= 'ausgeschaltet';
			IQ_stUniAnstgHMI.stHandFktHMI[2].sText:= 'einschalten';
   END_IF
	IF stUniAnstgFkt.nHandStat = 2	(*Handfunktion.2 aktiv*)
		THEN		 
			IQ_stUniAnstgHMI.stHandFktHMI[1].sColour:= cDefaultAsString;
			IQ_stUniAnstgHMI.stHandFktHMI[2].sColour:= cGruenAsString;
			IQ_stUniAnstgHMI.stHandFktHMI[1].sText:= 'ausschalten';
			IQ_stUniAnstgHMI.stHandFktHMI[2].sText:= 'eingeschaltet';
   END_IF
	IQ_stUniAnstgHMI.stHandFktHMI[3].sColour:= cDefaultAsString;
	IQ_stUniAnstgHMI.stHandFktHMI[3].sText:= ' ';
	IQ_stUniAnstgHMI.stHandFktHMI[4].sColour:= cDefaultAsString;
	IQ_stUniAnstgHMI.stHandFktHMI[4].sText:= ' ';
	IF bUmrFehl
		THEN
			IQ_stUniAnstgHMI.stHandFktHMI[5].sColour:= cOrangeAsString;
			IQ_stUniAnstgHMI.stHandFktHMI[5].sText:= 'Reset';
		ELSE
			IQ_stUniAnstgHMI.stHandFktHMI[5].sColour:= cBlauAsString;
			IQ_stUniAnstgHMI.stHandFktHMI[5].sText:= 'Reset';
   END_IF
	IF stUniAnstgFkt.nHandStat = 256	(*Funktion gesperrt*)
		THEN
			IQ_stUniAnstgHMI.stHandFktHMI[1].sText:= 'ausgeschaltet';
			IQ_stUniAnstgHMI.stHandFktHMI[2].sText:= 'einschalten';
			IQ_stUniAnstgHMI.stHandFktHMI[1].sColour:= cDefaultAsString;
			IQ_stUniAnstgHMI.stHandFktHMI[2].sColour:= cDefaultAsString;
			IQ_stUniAnstgHMI.stHandFktHMI[1].sColour:=
			IQ_stUniAnstgHMI.stHandFktHMI[2].sColour:=cDefaultAsString;
			IQ_stUniAnstgHMI.stHandFktHMI[1].byStatus:=
			IQ_stUniAnstgHMI.stHandFktHMI[2].byStatus:=
			IQ_stUniAnstgHMI.stHandFktHMI[3].byStatus:=
			IQ_stUniAnstgHMI.stHandFktHMI[4].byStatus:=
			IQ_stUniAnstgHMI.stHandFktHMI[5].byStatus:= 1;
		ELSE
			IQ_stUniAnstgHMI.stHandFktHMI[1].byStatus.0	:= I_bVerrHdFktZ;
			IQ_stUniAnstgHMI.stHandFktHMI[2].byStatus.0	:= I_bVerrHdFktV;
			IQ_stUniAnstgHMI.stHandFktHMI[3].byStatus:=
			IQ_stUniAnstgHMI.stHandFktHMI[4].byStatus:=
			IQ_stUniAnstgHMI.stHandFktHMI[5].byStatus:= 0;
   END_IF

2:	(*Antriebstyp Transport*) 
	
	IF GETBIT32 (TO_DWORD(stUniAnstgFkt.nHandStat), 0)	(*Handfunktion.1 aktiv*)
		THEN
			IQ_stUniAnstgHMI.stHandFktHMI[1].sColour:= cGruenAsString;
			IQ_stUniAnstgHMI.stHandFktHMI[1].sText:= 'ausschalten';
		ELSE
			IQ_stUniAnstgHMI.stHandFktHMI[1].sColour:= cDefaultAsString;
			IQ_stUniAnstgHMI.stHandFktHMI[1].sText:= 'zurück';
			IF GETBIT32 (TO_DWORD(stUniAnstgFkt.nHandStat), 1) THEN
				IQ_stUniAnstgHMI.stHandFktHMI[1].sText:= ' ';
			END_IF
   END_IF
	IF GETBIT32 (TO_DWORD(stUniAnstgFkt.nHandStat), 1)	(*Handfunktion.2 aktiv*)
		THEN		 
			IQ_stUniAnstgHMI.stHandFktHMI[2].sColour:= cGruenAsString;
			IQ_stUniAnstgHMI.stHandFktHMI[2].sText:= 'ausschalten';
		ELSE
			IQ_stUniAnstgHMI.stHandFktHMI[2].sColour:= cDefaultAsString;
			IQ_stUniAnstgHMI.stHandFktHMI[2].sText:= 'vor';
			IF GETBIT32 (TO_DWORD(stUniAnstgFkt.nHandStat), 0) THEN
				IQ_stUniAnstgHMI.stHandFktHMI[2].sText:= ' ';
			END_IF
   END_IF
	IF GETBIT32 (TO_DWORD(stUniAnstgFkt.nHandStat), 2)	(*Handfunktion.3 aktiv*)
		AND (GETBIT32 (TO_DWORD(stUniAnstgFkt.nHandStat), 0)
		OR   GETBIT32 (TO_DWORD(stUniAnstgFkt.nHandStat), 1))	 
		THEN
			IQ_stUniAnstgHMI.stHandFktHMI[3].sColour:= cGruenAsString;
			IQ_stUniAnstgHMI.stHandFktHMI[3].sText:= 'V = Nmin';
		ELSE
			IQ_stUniAnstgHMI.stHandFktHMI[3].sColour:= cDefaultAsString;
			IQ_stUniAnstgHMI.stHandFktHMI[3].sText:= 'V = Nmin';
   END_IF
	IF GETBIT32 (TO_DWORD(stUniAnstgFkt.nHandStat), 3)	(*Handfunktion.4 aktiv*)
		AND (GETBIT32 (TO_DWORD(stUniAnstgFkt.nHandStat), 0)
		OR   GETBIT32 (TO_DWORD(stUniAnstgFkt.nHandStat), 1))	 
		THEN
			IQ_stUniAnstgHMI.stHandFktHMI[4].sColour:= cGruenAsString;
			IQ_stUniAnstgHMI.stHandFktHMI[4].sText:= 'V = Nmax';
		ELSE
			IQ_stUniAnstgHMI.stHandFktHMI[4].sColour:= cDefaultAsString;
			IQ_stUniAnstgHMI.stHandFktHMI[4].sText:= 'V = Nmax';
   END_IF
	IF bUmrFehl
		THEN
			IQ_stUniAnstgHMI.stHandFktHMI[5].sColour:= cOrangeAsString;
			IQ_stUniAnstgHMI.stHandFktHMI[5].sText:= 'Reset';
		ELSE
			IQ_stUniAnstgHMI.stHandFktHMI[5].sColour:= cBlauAsString;
			IQ_stUniAnstgHMI.stHandFktHMI[5].sText:= 'Reset';
   END_IF
	IF stUniAnstgFkt.nHandStat = 256	(*Funktion gesperrt*)
		THEN
			IQ_stUniAnstgHMI.stHandFktHMI[1].sText:= 'zurück';
			IQ_stUniAnstgHMI.stHandFktHMI[2].sText:= 'vor';
			IQ_stUniAnstgHMI.stHandFktHMI[1].byStatus:=
			IQ_stUniAnstgHMI.stHandFktHMI[2].byStatus:=
			IQ_stUniAnstgHMI.stHandFktHMI[3].byStatus:=
			IQ_stUniAnstgHMI.stHandFktHMI[4].byStatus:=
			IQ_stUniAnstgHMI.stHandFktHMI[5].byStatus:= 1;
		ELSE
			IQ_stUniAnstgHMI.stHandFktHMI[1].byStatus.0	:= I_bVerrHdFktZ;
			IQ_stUniAnstgHMI.stHandFktHMI[2].byStatus.0	:= I_bVerrHdFktV;
			IQ_stUniAnstgHMI.stHandFktHMI[3].byStatus:=
			IQ_stUniAnstgHMI.stHandFktHMI[4].byStatus:=
			IQ_stUniAnstgHMI.stHandFktHMI[5].byStatus:= 0;
   END_IF

3:	(*Antriebstyp Verstellg.*)
	
	IQ_stUniAnstgHMI.stHandFktHMI[1].iDisplayMode	:= 0;
	IF GETBIT32 (TO_DWORD(stUniAnstgFkt.nHandStat), 0)	// Taste 1 für zurückfahren
		THEN
			IF NOT I_bEndlHdFktV
			THEN	// Verstellantrieb ist in Endlage
				IQ_stUniAnstgHMI.stHandFktHMI[1].sColour	:= cGruenAsString;
				IQ_stUniAnstgHMI.stHandFktHMI[1].sText		:= 'zurückgefahren';
			ELSE	// Verstellantrieb ist noch unterwegs
				IQ_stUniAnstgHMI.stHandFktHMI[1].iDisplayMode	:= 2;	// schnell blinken
				IQ_stUniAnstgHMI.stHandFktHMI[1].sColour:= cGelbAsString;
				IQ_stUniAnstgHMI.stHandFktHMI[1].sText:= 'zurückfahren';
			END_IF
		ELSE
			IF NOT I_bEndlHdFktZ 
			THEN
				IQ_stUniAnstgHMI.stHandFktHMI[1].sColour:= cGruenAsString;
				IQ_stUniAnstgHMI.stHandFktHMI[1].sText:= 'zurückgefahren';
			ELSE
				IQ_stUniAnstgHMI.stHandFktHMI[1].sColour:= cDefaultAsString;
				IQ_stUniAnstgHMI.stHandFktHMI[1].sText:= 'zurückfahren';
			END_IF
   END_IF
	
	IQ_stUniAnstgHMI.stHandFktHMI[2].iDisplayMode	:= 0;
	IF GETBIT32 (TO_DWORD(stUniAnstgFkt.nHandStat), 1)	// Taste 2 für vorfahren
		THEN
			IF NOT I_bEndlHdFktV
			THEN	// Verstellantrieb ist in Endlage
				IQ_stUniAnstgHMI.stHandFktHMI[2].sColour	:= cGruenAsString;
				IQ_stUniAnstgHMI.stHandFktHMI[2].sText		:= 'vorgefahren';
			ELSE	// Verstellantrieb ist noch unterwegs
				IQ_stUniAnstgHMI.stHandFktHMI[2].sColour	:= cGelbAsString;
				IQ_stUniAnstgHMI.stHandFktHMI[2].iDisplayMode	:= 2;	// schnell blinken
				IQ_stUniAnstgHMI.stHandFktHMI[2].sText		:= 'vorfahren';
			END_IF
		ELSE
			IF NOT I_bEndlHdFktV
			THEN
				IQ_stUniAnstgHMI.stHandFktHMI[2].sColour:= cGruenAsString;
				IQ_stUniAnstgHMI.stHandFktHMI[2].sText:= 'vorgefahren';
			ELSE
				IQ_stUniAnstgHMI.stHandFktHMI[2].sColour:= cDefaultAsString;
				IQ_stUniAnstgHMI.stHandFktHMI[2].sText:= 'vorfahren';
			END_IF
   END_IF
	
	IF GETBIT32 (TO_DWORD(stUniAnstgFkt.nHandStat), 2)	// Taste 3 für langsam
		THEN
			IQ_stUniAnstgHMI.stHandFktHMI[3].sColour:= cGruenAsString;
			IQ_stUniAnstgHMI.stHandFktHMI[3].sText:= 'langsam';
		ELSE
			IQ_stUniAnstgHMI.stHandFktHMI[3].sColour:= cDefaultAsString;
			IQ_stUniAnstgHMI.stHandFktHMI[3].sText:= 'langsam';
   END_IF
	IF GETBIT32 (TO_DWORD(stUniAnstgFkt.nHandStat), 3)	// Taste 4 für schnell
		THEN
			IQ_stUniAnstgHMI.stHandFktHMI[4].sColour:= cGruenAsString;
			IQ_stUniAnstgHMI.stHandFktHMI[4].sText:= 'schnell';
		ELSE
			IQ_stUniAnstgHMI.stHandFktHMI[4].sColour:= cDefaultAsString;
			IQ_stUniAnstgHMI.stHandFktHMI[4].sText:= 'schnell';
   END_IF
	
	IF bUmrFehl
		THEN
			IQ_stUniAnstgHMI.stHandFktHMI[5].sColour:= cOrangeAsString;
			IQ_stUniAnstgHMI.stHandFktHMI[5].sText:= 'Reset';
		ELSE
			IQ_stUniAnstgHMI.stHandFktHMI[5].sColour:= cBlauAsString;
			IQ_stUniAnstgHMI.stHandFktHMI[5].sText:= 'Reset';
   END_IF
	
	IF stUniAnstgFkt.nHandStat = 256	(*Funktion gesperrt*)
		THEN
			IF NOT I_bEndlHdFktZ 
			THEN
				IQ_stUniAnstgHMI.stHandFktHMI[1].sColour:= cGruenAsString;
				IQ_stUniAnstgHMI.stHandFktHMI[1].sText:= 'zurückgefahren';
			ELSE
				IQ_stUniAnstgHMI.stHandFktHMI[1].sColour:= cDefaultAsString;
				IQ_stUniAnstgHMI.stHandFktHMI[1].sText:= 'zurückfahren';
			END_IF
			IF NOT I_bEndlHdFktV 
			THEN
				IQ_stUniAnstgHMI.stHandFktHMI[2].sColour:= cGruenAsString;
				IQ_stUniAnstgHMI.stHandFktHMI[2].sText:= 'vorgefahren';
			ELSE
				IQ_stUniAnstgHMI.stHandFktHMI[2].sColour:= cDefaultAsString;
				IQ_stUniAnstgHMI.stHandFktHMI[2].sText:= 'vorfahren';
			END_IF
			IQ_stUniAnstgHMI.stHandFktHMI[3].sText:= 'langsam';
			IQ_stUniAnstgHMI.stHandFktHMI[4].sText:= 'schnell';
			IQ_stUniAnstgHMI.stHandFktHMI[1].byStatus:=
			IQ_stUniAnstgHMI.stHandFktHMI[2].byStatus:=
			IQ_stUniAnstgHMI.stHandFktHMI[3].byStatus:=
			IQ_stUniAnstgHMI.stHandFktHMI[4].byStatus:=
			IQ_stUniAnstgHMI.stHandFktHMI[5].byStatus:= 1;
		ELSE
			IQ_stUniAnstgHMI.stHandFktHMI[1].byStatus.0	:= I_bVerrHdFktZ;
			IQ_stUniAnstgHMI.stHandFktHMI[2].byStatus.0	:= I_bVerrHdFktV;
			IQ_stUniAnstgHMI.stHandFktHMI[3].byStatus:=
			IQ_stUniAnstgHMI.stHandFktHMI[4].byStatus:=
			IQ_stUniAnstgHMI.stHandFktHMI[5].byStatus:= 0;
   END_IF

4: (*Antriebstyp EilSchleich*)
	
	IF stUniAnstgFkt.nHandStat = 1	(*Handfunktion.1 aktiv*)
		THEN
			IQ_stUniAnstgHMI.stHandFktHMI[1].sColour:= cGruenAsString;
			IQ_stUniAnstgHMI.stHandFktHMI[1].sText:= 'negativ fahren';
		ELSE
			IQ_stUniAnstgHMI.stHandFktHMI[1].sColour:= cDefaultAsString;
			IQ_stUniAnstgHMI.stHandFktHMI[1].sText:= 'negativ fahren';
   END_IF
	IF stUniAnstgFkt.nHandStat = 2	(*Handfunktion.2 aktiv*)
		THEN		 
			IQ_stUniAnstgHMI.stHandFktHMI[2].sColour:= cGruenAsString;
			IQ_stUniAnstgHMI.stHandFktHMI[2].sText:= 'positiv fahren';
		ELSE
			IQ_stUniAnstgHMI.stHandFktHMI[2].sColour:= cDefaultAsString;
			IQ_stUniAnstgHMI.stHandFktHMI[2].sText:= 'positiv fahren';
   END_IF
	IQ_stUniAnstgHMI.stHandFktHMI[3].sColour:= cDefaultAsString;
	IQ_stUniAnstgHMI.stHandFktHMI[3].sText:= ' ';
	IQ_stUniAnstgHMI.stHandFktHMI[4].sColour:= cDefaultAsString;
	IQ_stUniAnstgHMI.stHandFktHMI[4].sText:= ' ';
	IF bUmrFehl
		THEN
			IQ_stUniAnstgHMI.stHandFktHMI[5].sColour:= cOrangeAsString;
			IQ_stUniAnstgHMI.stHandFktHMI[5].sText:= 'Reset';
		ELSE
			IQ_stUniAnstgHMI.stHandFktHMI[5].sColour:= cBlauAsString;
			IQ_stUniAnstgHMI.stHandFktHMI[5].sText:= 'Reset';
   END_IF
	IF stUniAnstgFkt.nHandStat = 256	(*Funktion gesperrt*)
		THEN
			IQ_stUniAnstgHMI.stHandFktHMI[1].sText:= 'negativ fahren';
			IQ_stUniAnstgHMI.stHandFktHMI[2].sText:= 'positiv fahren';
			IQ_stUniAnstgHMI.stHandFktHMI[1].sColour:=
			IQ_stUniAnstgHMI.stHandFktHMI[2].sColour:=cDefaultAsString;
			IQ_stUniAnstgHMI.stHandFktHMI[1].byStatus:=
			IQ_stUniAnstgHMI.stHandFktHMI[2].byStatus:=
			IQ_stUniAnstgHMI.stHandFktHMI[3].byStatus:=
			IQ_stUniAnstgHMI.stHandFktHMI[4].byStatus:=
			IQ_stUniAnstgHMI.stHandFktHMI[5].byStatus:= 1;
		ELSE
			IQ_stUniAnstgHMI.stHandFktHMI[1].byStatus.0	:= I_bVerrHdFktZ;
			IQ_stUniAnstgHMI.stHandFktHMI[2].byStatus.0	:= I_bVerrHdFktV;
			IQ_stUniAnstgHMI.stHandFktHMI[3].byStatus:=
			IQ_stUniAnstgHMI.stHandFktHMI[4].byStatus:=
			IQ_stUniAnstgHMI.stHandFktHMI[5].byStatus:= 0;
   END_IF
	
   END_CASE

	(**************************************************)
END_ACTION

ACTION z_FehlerAusw:


IF	nFehlercode <> 0
	AND bUmrFehl
THEN	
	CASE	nFehlercode  OF
		0:sFehlerstring:='Kein Fehler';
		1:sFehlerstring:='Überstrom';
		3:sFehlerstring:='Erdschluss';
		4:sFehlerstring:='Brems- Chopper';
		6:sFehlerstring:='NetzPhasen- ausfall';
		7:sFehlerstring:='Zwischenkreis- Überspannung';
		8:sFehlerstring:='Drehzahl-Überwachung';
		9:sFehlerstring:='Inbetriebnahme';
		10:sFehlerstring:='IPOS-ILLOP';
		11:sFehlerstring:='Übertemperatur';
		14:sFehlerstring := 'Geberfehler';
		17:sFehlerstring:='Systemstörung';
		18:sFehlerstring:='Systemstörung';
		19:sFehlerstring:='Systemstörung';
		20:sFehlerstring:='Systemstörung';
		21:sFehlerstring:='Systemstörung';
		22:sFehlerstring:='Systemstörung';
		23:sFehlerstring:='Systemstörung';
		24:sFehlerstring:='Systemstörung';
		25:sFehlerstring:='EEPROM';
		26:sFehlerstring:='Externe Klemme';
		29:sFehlerstring:= 'Endschalter angefahren';
		31:sFehlerstring:='TF/TH-Auslöser';
		32:sFehlerstring:='IPOS-Index- Überlauf';
		34:sFehlerstring:='Rampen- Timeout';
		35:sFehlerstring:='Betriebsart Ex-e-Schutz';
		36:sFehlerstring:='Option fehlt';
		37:sFehlerstring:='System- Watchdog';
		38:sFehlerstring:='System- Software';
		42: sFehlerstring := 'Schleppfehler';
		43:sFehlerstring:='RS485 Timeout';
		44:sFehlerstring:='Geräte- auslastung';
		45:sFehlerstring:='Initialisierung';
		47:sFehlerstring:='Systembus 1 Timeout';
		77:sFehlerstring:='IPOS-Steuer wort';
		78: sFehlerstring:= 'Software-Endschalter angefahren';
		80:sFehlerstring:='RAM-Test';
		81:sFehlerstring:='Startbedingung';
		82:sFehlerstring:='Ausgang offen';
		84:sFehlerstring:='Motorschutz';
		94:sFehlerstring:='Prüfsumme EEPROM';
		97:sFehlerstring:='Kopierfehler';
		98:sFehlerstring:='CRC Error Flash';
		100:sFehlerstring:='Schwingung/W arnung';
		101:sFehlerstring:='Schwingung Fehler';
		102:sFehlerstring:='Ölalterung/ Warnung';
		103:sFehlerstring:='Ölalterung/ Fehler';
		104:sFehlerstring:='Ölalterung/ Übertempe- ratur';
		105:sFehlerstring:='Ölalterung/ Bereitmeldung';
		106:sFehlerstring:='Bremsver- schleiß';
		110:sFehlerstring:='Ex-e-Schutz';
		111:sFehlerstring:='Systembus (SBus) Fehler';
		113:sFehlerstring:='Drahtbruch Analogeingang';
		116:sFehlerstring:='Fehler Applikationsmodul Subfehler:'; 
	END_CASE
ELSE
	sFehlerstring := '';
END_IF
END_ACTION

ACTION z_FehlMeld:

	(**************************************************)	
	(*Meldungen ausgeben*)

	IQ_stUniAnstgHMI.stMeldAusgHMI.SourceID			:= 0;	// Nicht mehr verwendet
	IQ_stUniAnstgHMI.stMeldAusgHMI.SourceName			:= I_sStatName;
	IQ_stUniAnstgHMI.stMeldAusgHMI.sAktorName			:= I_sAktorName;
	
	IF I_sAktorBMK <> ''
	THEN	// I_sAktorBMK ist beschrieben. Damit wird der String als BMK genommen
		IQ_stUniAnstgHMI.stMeldAusgHMI.sBMK	:= I_sAktorBMK;
	ELSE	// Der Kommentar von VARINFO wird als BMK genommen
		IQ_stUniAnstgHMI.stMeldAusgHMI.sBMK	:= I_stVarInfoBMK.Comment;
	END_IF

	// Meldung: FU nicht Betriebsbereit
	tonMeldNichtBtb(
		IN:= (arrAntrGruppeFrg[I_nSchutzBer]
				AND (NOT bUmrStat
					OR NOT bDatenFrg
					OR bUmrFehl)
				AND bVersEingAusgSchaltsOk),
		PT:= t#2s);
	IQ_stUniAnstgHMI.stMeldAusgHMI.bMeldNichtBtb		:= tonMeldNichtBtb.Q
																		OR bTestMeldAntr;

	// Meldung: FU wurde ggf. im Schaltschrank gesperrt. Meldung verzögern, weil das Bit bEndstFrg erst verspätet TRUE wird.
	tonMeldUmrichterGesperrt(
		IN	:= bUmrStat
				AND bDatenFrg
				AND NOT bEndstFrg
				AND (stUniAnstgFkt.arrFktAusfg[1]
					OR stUniAnstgFkt.arrFktAusfg[0]),
		PT	:= T#250MS,
	);

	IF tonMeldUmrichterGesperrt.Q
	THEN
		bUmrichterGesperrt := TRUE;
	ELSIF	bEndstFrg
	THEN
		bUmrichterGesperrt := FALSE;
	END_IF
IQ_stUniAnstgHMI.stMeldAusgHMI.bMeldUmrichterGesperrt	:= bUmrichterGesperrt;
	
tonVerzFehlerstring(
	IN := sFehlerstring <> ''
				AND sLetzerFehlerstring = sLetzerFehlerstring,
	PT := t#500MS
);

	IF sFehlerstring <> ''
	THEN
		IQ_stUniAnstgHMI.stMeldAusgHMI.bMeldFehlercode 				:= tonVerzFehlerstring.Q;
		IQ_stUniAnstgHMI.stMeldAusgHMI.sMeldUmrichterfehler		:= sFehlerstring;
	ELSE
		IQ_stUniAnstgHMI.stMeldAusgHMI.bMeldFehlercode			 	:= FALSE;
		IQ_stUniAnstgHMI.stMeldAusgHMI.sMeldUmrichterfehler		:= '';
	END_IF

	sLetzerFehlerstring := sFehlerstring;

	IF I_eAntriebTyp = eEilSchleich
	THEN
		IQ_stUniAnstgHMI.stMeldAusgHMI.bMeldNichtReferenz		:= (NOT I_RefAchse.stStatus.bInReferz
																					AND NOT I_RefAchse.stGrdfkt.bRefrz_ausf)
																					OR bTestMeldAntrEilSchleich;
		IQ_stUniAnstgHMI.stMeldAusgHMI.bMeldReffahrtStart		:= I_RefAchse.stGrdfkt.bRefrz_ausf
																					OR bTestMeldAntrEilSchleich;
	END_IF

	IF I_eAntriebTyp = eVerstellg
	THEN
		tonMeldLaufzeit0(	IN := stUniAnstgFkt.arrHandFkt[0]
										AND NOT I_bEndlHdFktZ,
								PT := I_tLaufzeitMeld);
		tonMeldLaufzeit1(	IN := stUniAnstgFkt.arrHandFkt[1]
										AND NOT I_bEndlHdFktV,
								PT := I_tLaufzeitMeld);
		IQ_stUniAnstgHMI.stMeldAusgHMI.bMeldLaufzeit0		:= tonMeldLaufzeit0.Q
																					OR bTestMeldAntrVerstellg;
		IQ_stUniAnstgHMI.stMeldAusgHMI.bMeldLaufzeit1		:= tonMeldLaufzeit1.Q
																					OR bTestMeldAntrVerstellg;
	END_IF
	
	
	(*Zus. Hinweise HF-Aggregate*)
	IF bTestMeldAntrHF
	THEN
		IQ_stUniAnstgHMI.stMeldAusgHMI.bMeldEinlZyklAktiv	:=
		IQ_stUniAnstgHMI.stMeldAusgHMI.bMeldEinlZyklBeendet:=
		IQ_stUniAnstgHMI.stMeldAusgHMI.bMeldWarmlaufZykl	:= TRUE;
	ELSIF nStepEinlZykl > 1 AND nStepEinlZykl < 300 
	THEN 						
		IQ_stUniAnstgHMI.stMeldAusgHMI.bMeldEinlZyklAktiv	:= TRUE;
		IQ_stUniAnstgHMI.stMeldAusgHMI.bMeldEinlZyklBeendet:=
		IQ_stUniAnstgHMI.stMeldAusgHMI.bMeldWarmlaufZykl	:= FALSE;
	ELSIF nStepEinlZykl = 300 
	THEN
		IQ_stUniAnstgHMI.stMeldAusgHMI.bMeldEinlZyklAktiv	:= FALSE;
		IQ_stUniAnstgHMI.stMeldAusgHMI.bMeldEinlZyklBeendet:= TRUE;
		IQ_stUniAnstgHMI.stMeldAusgHMI.bMeldWarmlaufZykl	:= FALSE;
	ELSIF (nStepBetrZykl > 1 AND nStepBetrZykl < 400)
      OR (nStepBetrZykl < 0) 
	THEN
		IQ_stUniAnstgHMI.stMeldAusgHMI.bMeldEinlZyklAktiv	:=
		IQ_stUniAnstgHMI.stMeldAusgHMI.bMeldEinlZyklBeendet:= FALSE;
		IQ_stUniAnstgHMI.stMeldAusgHMI.bMeldWarmlaufZykl	:= TRUE;
	ELSE							
		IQ_stUniAnstgHMI.stMeldAusgHMI.bMeldEinlZyklAktiv	:=
		IQ_stUniAnstgHMI.stMeldAusgHMI.bMeldEinlZyklBeendet:=
		IQ_stUniAnstgHMI.stMeldAusgHMI.bMeldWarmlaufZykl	:= FALSE;
	END_IF
END_ACTION

END_FUNCTION_BLOCK

// POUs/UniBausteine/FB_UniAntrAnstgSEW_IO
(*
Beschreibung :	SEW-FU-Steuerung für die Verwendung von IO's also über Hardware Ein- und Ausgänge.
					Nicht über Prozessabbild wie mit der FSE24B. Auch eine Warmlaufphase für Bohraggregate wäre möglich, wenn die Ausgänge verdrahtet sind.
					inkl. Handling - Handfunktinen
										- Meldefunktionen
										- Betriebsarten
										- Schutzbereiche
					Datentypen: ST_UniBaustein
									ST_UniAntrAnstg
									ST_NcAchsen
									Tc2_MC2.AXIS_REF
					Ressourcen: GlobalVar_Allgemein
									GlobalVar_Farben
									AllgemeineParameter
TwinCat Vers.:	3.1.4024.40							
*)
FUNCTION_BLOCK FB_UniAntrAnstgSEW_IO
VAR_INPUT

	I_sSchaltSchr		:Tc2_System.T_MaxString;	// Aktueller Schaltschrank in dem der FU sitzt
	I_sStatName			:Tc2_System.T_MaxString;	// Aktueller Stationsname in dem der Motor sitzt
	I_sAktorName		:Tc2_System.T_MaxString;	// Aktueller Aktorname von der Funktion des Motors
	I_sAktorBMK			:Tc2_System.T_MaxString;	// BMK vom FU

	I_bResHandFkt		:BOOL;						// Funktion-Reset für Grundstellungsablauf. Alle Zuweisungen aus
	I_arrZuwGrdstFkt	:ARRAY[0..3] OF BOOL;	// Funktion-Zuweisung Grundstellungsablauf: 0:Richtungsvorgabe zurück, 1:Richtungsvorgabe vor, 2: (N11), 3: (N12), 2&3 zusammen (N13)
	I_arrZuwAutomFkt	:ARRAY[0..3] OF BOOL;	// Funktion-Zuweisung Automatikablauf: 0:Richtungsvorgabe zurück, 1:Richtungsvorgabe vor, 2: (N11), 3: (N12), 2&3 zusammen (N13)

	I_bUmrStat			:BOOL;	// Umrichterstatus als Hardwareeingang

	I_eAntriebTyp		:E_AntriebTyp;	// Antriebsfunktion

	I_RefAchse			:REFERENCE TO ST_NcAchsen;	// Verweis zur arrNcAchsen-Strucktur. Bei einer Eil-Schleichachse einfach zuweisen.
	I_RefAxis			:REFERENCE TO Tc2_MC2.AXIS_REF;	// Verweis zur arrAxisRef-Strucktur. Bei einer Eil-Schleichachse einfach zuweisen.

	I_nAntrEinsGrp		:INT;		// Aktuelle Netzeinschaltgruppe
	I_nSchutzBer		:INT;		// Schutzbereich => Betriebsart

	// Optional /Antriebstyp Aggregat
	I_bResHdBetr		:BOOL;	// Auschalten des Motors beim Wechsel auf Handbetrieb
	// Optional /Antriebstyp Transport/Verstellung
	I_bVerrHdFktV		:BOOL;	// Sperren Handfunktion Richtung Vor	
	I_bVerrHdFktZ		:BOOL;	// Sperren Handfunktion Richtung Zurück
	// Optional /Antriebstyp Verstellung/Antriebstyp EilSchleich
	I_bEndlHdFktV		:BOOL;	// Endlage Sensor Richtung Vor		
	I_bEndlHdFktZ		:BOOL;	// Endlage Sensor Richtung Zurück	
	I_bVerzHdFktV		:BOOL;	// Verzögerung Sensor Richtung Vor	
	I_bVerzHdFktZ		:BOOL;	// Verzögerung Sensor Richtung Zurück

	I_bExtReglFrg		:BOOL:= TRUE; // Externes Freigabesignal

	I_bAnwEinlZykl		:BOOL;	// Anwahl Erstinbetriebn.-Einlaufzyklus

	I_bStandbyBetr		:BOOL;	// Antrieb im Standby-Betrieb. Kann statt I_arrZuwAutomFkt[1] zur Hochlaufphase genutzt werden.
	
	I_tLaufzeitMeld	:TIME := T#10S; // Zeit bis zur Laufzeitmeldung

{attribute 'hide'}
	I_arrBetrZyklPhase:ARRAY[1..4] OF TIME	:= [T#1M,T#1M,T#1M,T#1M];	// Zeiten für das Warmlauf im Betrieb 1-3 ist Warmlaufen 4 ist Warmhalten
{attribute 'hide'}	
	I_tPause				:TIME := T#15M;
	
	I_stVarInfoBMK		:__SYSTEM.VAR_INFO;	// Optional: __VARINFO von dem Hardwareeingang I_stSEWInput oder I_stSEWOutput. Kann I_sAktorBMK ersetzen. I_sAktorBMK ist aber dominant. Nicht im Aufruf verwenden => separate Zuweisung
END_VAR
VAR_IN_OUT

	IQ_stUniAnstgHMI	:ST_UniAntrAnstg;	// HMI-Strukturen

END_VAR
VAR_OUTPUT

	Q_bAbfrStatUmr		:BOOL;	// Statusabfrage Umrichter; ist bei diesem Baustein einfach eine Weiterleitung der Eingangsvariable für den Umrichter

	Q_bAnstNetzUmr		:BOOL;	// Netzansteuerung Umrichter
	Q_bAnstReglFrg		:BOOL;	// Reglerfreigabe Umrichter
	
	Q_bRichtVrgV		:BOOL;	// Richtungsfreigabe Vorwärts über Ausgang. Langsame geschwindigkeit, wenn nicht Q_bSollwVrg angewählt. Bei Aggregat mit Hochlaufphase = 33% bzw. Leerlaufdrehzahl
	Q_bRichtVrgR		:BOOL;	// Richtungsfreigabe Rückwärts über Ausgang. Langsame geschwindigkeit, wenn nicht Q_bSollwVrg angewählt
	Q_bSollwVrg_N11	:BOOL;	// Sollwertvorwahl N11 über Ausgang. Standardmäßig nur bei Transporten verdrahtet. Bei Aggregat mit Hochlaufphase = 66%
	Q_bSollwVrg_N12	:BOOL;	// Sollwertvorwahl N12 über Ausgang. Nur für Aggregate mit Warmlaufphasen sinnvoll. Bei Aggregat mit Hochlaufphase = 100%

END_VAR
VAR
																						
	rtrigHandFkt0		:R_TRIG;
	rtrigHandFkt1		:R_TRIG;												
	rtrigHandFkt2		:R_TRIG;
	rtrigHandFkt3		:R_TRIG;

	bEndstFrg			:BOOL;
	bUmrStat				:BOOL;

	tonDrehzNnull		:TON;
	tonDrehzNnenn		:TON;
	
	tonMeldLaufzeit0	:TON;
	tonMeldLaufzeit1	:TON;
	
	//Relevante Variablen zur Diagnose
	stUniAnstgFkt		:ST_UniBaustein;

	//Zus. Variablen Betrieb HF-Aggregate
	nStepEinlZykl		:INT;
	nEinlZyklPhase		:INT;
	tonEinlZyklPhase	:TON;
	arrEinlZyklPhase	:ARRAY[1..21] OF TIME := [T#1M, T#2M, T#1M, T#2M, T#1M, T#2M, T#1M, T#2M, T#1M, T#2M, T#1M, T#2M, T#1M, T#2M, T#1M, T#2M, T#30M, T#5M, T#30M, T#5M];
	arrEinlZyklDrehz	:ARRAY[1..21] OF BYTE:= [1, 0, 1, 0, 1, 0, 2, 0, 2, 0, 2, 0, 3, 0, 3, 0, 3, 0, 3, 0];	// Bitweises auflösen der Ausgänge für die Geschwindigkeiten mit Richtungsfreigabe, N11 und N12

	nStepBetrZykl		:INT;
	nBetrZyklPhase		:INT;
	tonBetrZyklPhase	:TON;
	nDrehzBetrZykl		:LREAL;

	bHochlZyklStart	:BOOL;
	bHochlZyklEnde		:BOOL;
END_VAR

	(*Uni.- Antriebsansteuerung /SEW-Umrichter(EtherCAT)*)
	
	(**************************************************)	
	(*Aufruf-Bereichskontrolle*)

	IF I_nSchutzBer <= 0 OR I_nSchutzBer > cAnzSchutzBer
		OR ((NOT __ISVALIDREF(I_RefAchse)
				OR NOT __ISVALIDREF(I_RefAxis))
			AND I_eAntriebTyp = E_AntriebTyp.eEilSchleich)
		OR	I_nAntrEinsGrp <= 0 OR I_nAntrEinsGrp > cAnzEinschGrp
		THEN
			IF I_nSchutzBer <= 0 OR I_nSchutzBer > cAnzSchutzBer
			THEN
				IQ_stUniAnstgHMI.stMeldAusgHMI.sMeldText		:= 'I_nSchutzBer = 0 oder zu gross.';
			ELSIF I_nAntrEinsGrp <= 0 OR I_nAntrEinsGrp > cAnzEinschGrp
			THEN
				IQ_stUniAnstgHMI.stMeldAusgHMI.sMeldText		:= 'I_nAntrEinsGrp = 0 oder zu gross.';
			ELSE
				IQ_stUniAnstgHMI.stMeldAusgHMI.sMeldText		:= 'I_RefAchse oder I_RefAxis nicht beschrieben.';
			END_IF
			
			IQ_stUniAnstgHMI.stMeldAusgHMI.SourceName			:= I_sStatName;
			IQ_stUniAnstgHMI.stMeldAusgHMI.sAktorName			:= I_sAktorName;
			
			IF I_sAktorBMK <> ''
			THEN
 				IQ_stUniAnstgHMI.stMeldAusgHMI.sBMK	:= I_sAktorBMK;
			ELSE
				IQ_stUniAnstgHMI.stMeldAusgHMI.sBMK	:= I_stVarInfoBMK.Comment;
			END_IF
			
			IQ_stUniAnstgHMI.stMeldAusgHMI.bMeldHinweis		:= TRUE;
			
			// Texte der Handfunktionen zuweisen. Das sieht sonst schieße aus in der HMI
			stUniAnstgFkt.nHandStat	:= 256;	// Funktion sperren
			y_ZustAnzg();
			
			RETURN;
		ELSE
			IQ_stUniAnstgHMI.stMeldAusgHMI.bMeldHinweis	:= FALSE;
			IQ_stUniAnstgHMI.stMeldAusgHMI.sMeldText		:= '';
	END_IF

	(**************************************************)	
	(*Haendling Uni-Struktur*)
	
	CASE I_eAntriebTyp OF
		 
1:	(*Antriebstyp Aggregat*)
	
	a_Aggregat();

2:	(*Antriebstyp Transport*) 
	
	b_Transport();

3:	(*Antriebstyp Verstellg.*)

	c_Verstellg();	

4: (*Antriebstyp EilSchleich*)	
	
	d_EilSchleich();
	
5:	(*Antriebstyp HF-Aggregat*)
	
	a_Aggregat();

	u_AggEinlZykl(); //Einlaufphasen HF-Aggregat 
	v_AggBetrZykl(); //Betriebphasen HF-Aggregat
	
   END_CASE
	
	(**************************************************)	
	(*EtherCAT-Anschaltung*)	

	w_InOutSEW();

	(**************************************************)	
	(*Ausgänge zuweisen*)

	x_AusgZuw();
	
	(**************************************************)	
	(*Zustände anzeigen*)

	y_ZustAnzg();

	(**************************************************)	
	(*Meldungen ausgeben*)

	z_FehlMeld();
	
	(**************************************************)

ACTION a_Aggregat:
	(*Antriebstyp "Aggregat" /z.B. FU-Bohr.-Fräsaggregate...*)

	(*Verwendete Softkeytasten = 5 (s.Beispiel)*)

   (*       "Handfunktion"       /   "Softkeytaste 1"   /   "Softkeytaste 2"   /   "Softkeytaste 3"   /   "Softkeytaste 4"   /   "Softkeytaste 5"   *)
	(*                                                                          															  								 *) 
   (*------- Bohraggregat -------/_____ausschalten______/_____einschalten______/_________Frei_________/_________Frei_________/________Reset_________*)

	(*Softkeyleiste.1		:Funktion ausschalten		*)
	(*Softkeyleiste.2		:Funktion einschalten		*)
	(*Softkeyleiste.3		:Platzhalter					*)
	(*Softkeyleiste.4		:Platzhalter					*)
	(*Softkeyleiste.5		:Platzhalter					*)

	(*Hinweis:
	- Funktion wird durch "ResHdBetr" bei Betriebsartenwechsel zurückgenommen
	*)

	(**************************************************)	

	stUniAnstgFkt.bHandAnw0:= IQ_stUniAnstgHMI.stHandFktHMI[1].bySwitch > 0;
	stUniAnstgFkt.bHandAnw1:= IQ_stUniAnstgHMI.stHandFktHMI[2].bySwitch > 0;	
	
	IF arrBetrartAutomAktiv[I_nSchutzBer]
		OR I_bResHandFkt
		OR NOT I_bExtReglFrg
		OR NOT arrAntrGruppeFrg[I_nSchutzBer]
		THEN
			stUniAnstgFkt.arrHandFkt[1]:= FALSE;
		ELSE
			IF arrBetrartAutomSpeichn[I_nSchutzBer]
				THEN
					IF NOT I_bResHdBetr THEN
						stUniAnstgFkt.arrHandFkt[1]:= stUniAnstgFkt.arrFktAusfg[1];
					END_IF
				ELSE
					IF NOT arrGrdstlgBetrAktiv[I_nSchutzBer]
						AND arrBetrartHandAktiv[I_nSchutzBer]
						THEN
							 IF stUniAnstgFkt.bHandAnw1 THEN
								 stUniAnstgFkt.arrHandFkt[1]:= TRUE;
							 END_IF
							 IF stUniAnstgFkt.bHandAnw0 THEN
								 stUniAnstgFkt.arrHandFkt[1]:= FALSE;
							 END_IF
					END_IF
			END_IF
	END_IF

	IF arrBetrartHandAktiv[I_nSchutzBer]
		THEN
			IF stUniAnstgFkt.arrHandFkt[1]
				THEN
					stUniAnstgFkt.nHandStat:= 2;	(*Handfunktion.2 aktiv*)
				ELSE
					stUniAnstgFkt.nHandStat:= 1;	(*Handfunktion.1 aktiv*)
			END_IF
		ELSE
			stUniAnstgFkt.nHandStat:= 256;		(*Funktion gesperrt*)
	END_IF

	(**************************************************)	

	IF arrBetrartHandAktiv[I_nSchutzBer]
		THEN
			stUniAnstgFkt.arrGrdstFkt[1]:= I_arrZuwGrdstFkt[1];
		ELSE
			stUniAnstgFkt.arrGrdstFkt[1]:= FALSE;
   END_IF
	IF arrBetrartAutomAktiv[I_nSchutzBer] OR TRUE //ToDo
		THEN
			stUniAnstgFkt.arrAutomFkt[1]:= I_arrZuwAutomFkt[1];
		ELSE
			stUniAnstgFkt.arrAutomFkt[1]:= FALSE;
   END_IF

	(**************************************************)	

	stUniAnstgFkt.arrFktAusfg[1]:= stUniAnstgFkt.arrGrdstFkt[1]
										 	 OR stUniAnstgFkt.arrHandFkt[1]
										 	 OR stUniAnstgFkt.arrAutomFkt[1];

	(**************************************************)
END_ACTION

ACTION b_Transport:
	(*Antriebstyp "Transport" /z.B. FU-Transportsegmente...*)

	(*Verwendete Softkeytasten = 5 (s.Beispiel)*)

   (*       "Handfunktion"       /   "Softkeytaste 1"   /   "Softkeytaste 2"   /   "Softkeytaste 3"   /   "Softkeytaste 4"   /   "Softkeytaste 5"   *)
	(*                                                                          															  								 *) 
	(*----- Transportantrieb -----/_einschalten (zurück)_/___einschalten (vor)__/_________N11__________/_________N12__________/_________Frei_________*)

	(*Softkeyleiste.1		:Funktion ein.-ausschalten Reversierend*)
	(*Softkeyleiste.2		:Funktion ein.-ausschalten             *)
	(*Softkeyleiste.3		:Funktion langsame Drehzahl (SollwMin) *)
	(*Softkeyleiste.4		:Funktion schnelle Drehzahl (SollwVrg) *)
	(*Softkeyleiste.5		:Platzhalter									 *)

	(*Hinweis:
	- Funktion wird durch "VerrHdFkt" gesperrt (z.B. kein Reversierbetrieb...)
	*)

	(**************************************************)	

	stUniAnstgFkt.bHandAnw0:= IQ_stUniAnstgHMI.stHandFktHMI[1].bySwitch > 0;
	stUniAnstgFkt.bHandAnw1:= IQ_stUniAnstgHMI.stHandFktHMI[2].bySwitch > 0;
	stUniAnstgFkt.bHandAnw2:= IQ_stUniAnstgHMI.stHandFktHMI[3].bySwitch > 0;
	stUniAnstgFkt.bHandAnw3:= IQ_stUniAnstgHMI.stHandFktHMI[4].bySwitch > 0;
	
	IF arrBetrartAutomAktiv[I_nSchutzBer]
		OR I_bResHandFkt
		OR NOT I_bExtReglFrg
		THEN
			stUniAnstgFkt.arrHandFkt[0]:=
			stUniAnstgFkt.arrHandFkt[1]:=
			stUniAnstgFkt.arrHandFkt[2]:=
			stUniAnstgFkt.arrHandFkt[3]:= FALSE;
		ELSE
			IF NOT arrBetrartAutomSpeichn[I_nSchutzBer]
				THEN
					IF NOT arrGrdstlgBetrAktiv[I_nSchutzBer]
						THEN
							// Vor
							rtrigHandFkt1 (CLK:= stUniAnstgFkt.bHandAnw1);
							IF rtrigHandFkt1.Q THEN
								stUniAnstgFkt.arrHandFkt[1]:= NOT stUniAnstgFkt.arrHandFkt[1];
							END_IF
							IF NOT arrBetrartHandAktiv[I_nSchutzBer]
								OR stUniAnstgFkt.arrHandFkt[0]
								OR I_bVerrHdFktV THEN
								stUniAnstgFkt.arrHandFkt[1]:= FALSE;
							END_IF

							// Zurück
							rtrigHandFkt0 (CLK:= stUniAnstgFkt.bHandAnw0);
							IF rtrigHandFkt0.Q THEN
								stUniAnstgFkt.arrHandFkt[0]:= NOT stUniAnstgFkt.arrHandFkt[0];
							END_IF
							IF NOT arrBetrartHandAktiv[I_nSchutzBer]
								OR stUniAnstgFkt.arrHandFkt[1]
							THEN
								stUniAnstgFkt.arrHandFkt[0]:= FALSE;
							END_IF

							// N11 umschalten
							rtrigHandFkt2 (CLK:= stUniAnstgFkt.bHandAnw2);
							IF rtrigHandFkt2.Q THEN
								stUniAnstgFkt.arrHandFkt[2]:= NOT stUniAnstgFkt.arrHandFkt[2];
							END_IF
							IF NOT arrBetrartHandAktiv[I_nSchutzBer]
								OR I_bVerrHdFktZ
								OR I_bVerrHdFktV THEN
								stUniAnstgFkt.arrHandFkt[2]:= FALSE;
							END_IF
							
							// N12 umschalten							
							rtrigHandFkt3 (CLK:= stUniAnstgFkt.bHandAnw3);
							IF rtrigHandFkt3.Q THEN
								stUniAnstgFkt.arrHandFkt[3]:= NOT stUniAnstgFkt.arrHandFkt[3];
							END_IF
							IF NOT arrBetrartHandAktiv[I_nSchutzBer]
								OR I_bVerrHdFktZ
								OR I_bVerrHdFktV THEN
								stUniAnstgFkt.arrHandFkt[3]:= FALSE;
							END_IF
					END_IF
			END_IF
	END_IF

	IF arrBetrartHandAktiv[I_nSchutzBer]
		THEN
			stUniAnstgFkt.nHandStat:= 0;			(*Funktion freigegeben*)
			IF stUniAnstgFkt.arrHandFkt[1]
				THEN
					stUniAnstgFkt.nHandStat:= 2;	(*Handfunktion.2 aktiv*)
			END_IF
			IF stUniAnstgFkt.arrHandFkt[0]
				THEN
					stUniAnstgFkt.nHandStat:= 1;	(*Handfunktion.1 aktiv*)
			END_IF
			IF stUniAnstgFkt.arrHandFkt[2]
				THEN
					stUniAnstgFkt.nHandStat:=
					stUniAnstgFkt.nHandStat + 8;	(*Handfunktion.4 aktiv*)
				ELSE
					stUniAnstgFkt.nHandStat:=
					stUniAnstgFkt.nHandStat + 4;	(*Handfunktion.3 aktiv*)
			END_IF
			IF stUniAnstgFkt.arrHandFkt[3]
				THEN
					stUniAnstgFkt.nHandStat:=
					stUniAnstgFkt.nHandStat + 8;	(*Handfunktion.4 aktiv*)
				ELSE
					stUniAnstgFkt.nHandStat:=
					stUniAnstgFkt.nHandStat + 4;	(*Handfunktion.3 aktiv*)
			END_IF
		ELSE
			stUniAnstgFkt.nHandStat:= 256;		(*Funktion gesperrt*)
	END_IF

	(**************************************************)	

